ORGANIZATION_BLOCK "HardwareInterrupt"   // OB40, SCL, HardwareInterrupt
{ S7_Optimized_Access := 'TRUE' }
// stored: SetENOAutomatically false
   VAR_INPUT
      LADDR : HW_IO;   // Hardware identifier
      USI : Word;   // User structure identifier
      IChannel : USInt;   // Interrupt channel number
      EventType : Byte;   // EventType
      PointAddr : DWord;
   END_VAR
BEGIN
   REGION Description head
       //==================================================================================
       // POSALUX Swiss SA / (C) Copyright 2025
       //----------------------------------------------------------------------------------
       // Title: Hardware interrupt
       // Comment/Function: Executes when a relevant hardware event occurs
       // Author: Fabien WALDT
       // Engineering: TIA Portal v19
       //----------------------------------------------------------------------------------
       // Change log table:
       // Version  | Date     | Expert in charge | Changes applied
       //----------------------------------------------------------------------------------
       // 00.00.01 | 20250423 | WFA              | First released version
       //==================================================================================
   END_REGION

   REGION NCK Process IRT
       "LBP_NCKProcessIRT"(Flags => NULL);
   END_REGION
END_ORGANIZATION_BLOCK

ORGANIZATION_BLOCK "IO_AccessError"   // OB122, SCL, IOAccessError
{ S7_Optimized_Access := 'TRUE' }
// stored: SetENOAutomatically false
   VAR_INPUT
      BlockNr : UInt;   // Number of causing block
      Reaction : USInt;   // 0:ignore, 1:substitute, 2:skip
      Fault_ID : Byte;   // 16#42:reading, 16#43:writing
      BlockType : USInt;   // 16#01:OB, 16#02:FC, 16#03:FB, 16#04:SFC, 16#05:SFB, 16#06:DB: Type of block causing the error
      Area : USInt;   // 16#81:I, 16#82:Q: IO area where the IOaccess error occured
      DBNr : DB_ANY;   // Reserved for system
      Csg_OBNr : OB_ANY;   // Number of OB causing the error
      Csg_Prio : USInt;   // Priority of OB causing the error
      Width : USInt;   // 0:bit, 1:byte, 2:word, 3:dword, 4:lword
   END_VAR
BEGIN
   REGION Description head
       //==================================================================================
       // POSALUX Swiss SA / (C) Copyright 2025
       //----------------------------------------------------------------------------------
       // Title: IO_AccessError
       // Comment/Function: Executes whenever an error occurs while accessing data on a module
       // Author: Fabien WALDT
       // Engineering: TIA Portal v19
       //----------------------------------------------------------------------------------
       // Change log table:
       // Version  | Date     | Expert in charge | Changes applied
       //----------------------------------------------------------------------------------
       // 00.00.01 | 20250423 | WFA              | First released version
       //==================================================================================
   END_REGION
END_ORGANIZATION_BLOCK

ORGANIZATION_BLOCK "RackOrStationFailure"   // OB86, SCL, RackOrStationFailure
{ S7_Optimized_Access := 'TRUE' }
// stored: SetENOAutomatically false
   VAR_INPUT
      LADDR : HW_DEVICE;   // Hardware identifier
      Event_Class : Byte;   // Event class
      Fault_ID : Byte;   // Fault identifier
   END_VAR
BEGIN
   REGION Description head
       //==================================================================================
       // POSALUX Swiss SA / (C) Copyright 2025
       //----------------------------------------------------------------------------------
       // Title: Main
       // Comment/Function: Executes when the CPU detects the failure
       //                   or communication loss of a distributed rack or station
       // Author: Fabien WALDT
       // Engineering: TIA Portal v19
       //----------------------------------------------------------------------------------
       // Change log table:
       // Version  | Date     | Expert in charge | Changes applied
       //----------------------------------------------------------------------------------
       // 00.00.01 | 20250423 | WFA              | First released version
       //==================================================================================
   END_REGION
END_ORGANIZATION_BLOCK

ORGANIZATION_BLOCK "Startup"   // OB100, SCL, Startup
TITLE = "Complete Restart"
{ S7_Optimized_Access := 'TRUE' }
// stored: SetENOAutomatically false
   VAR_INPUT
      LostRetentive : Bool;   // True if retentive data are lost
      LostRTC : Bool;   // True if date and time are lost
   END_VAR
   VAR_TEMP
      tLastDateTime : DTL;
      tLasDateTimeSec : DInt;
      tActualDateTime : DTL;
      tActualDateTimeINT : DInt;
      tActualDateTimeSec : DInt;
   END_VAR
BEGIN
   REGION Description head
       //==================================================================================
       // POSALUX Swiss SA / (C) Copyright 2025
       //----------------------------------------------------------------------------------
       // Title: Startup
       // Comment/Function: Executes one time when the operating mode of the CPU changes from STOP to RUN
       // Author: Fabien WALDT
       // Engineering: TIA Portal v19
       //----------------------------------------------------------------------------------
       // Change log table:
       // Version  | Date     | Expert in charge | Changes applied
       //----------------------------------------------------------------------------------
       // 00.00.01 | 20250423 | WFA              | First released version
       //==================================================================================
   END_REGION

   REGION Safety Brake Test
       "LBP_AlarmMsgs".UserA[5].A70UUxx[12] := FALSE;  // Msg 700512 "SAFETY : THE BRAKE TEST IS NOT WORKING, PLEASE RESET"
   END_REGION

   REGION Config NC Panel
       "LBP_ConfigBP"(MCPNum := "LBP_ConfigData".MCPNum,
                      MCP1In := "MCP1_In",
                      MCP1Out := "MCP1_Out",
                      MCP1BusAdr := "LBP_ConfigData".MCP1BusAdr,
                      MCP1Timeout := "LBP_ConfigData".MCP1Timeout,
                      MCP2In := NULL,
                      MCP2Out := NULL,
                      MCP2BusAdr := "LBP_ConfigData".MCP2BusAdr,
                      MCP2Timeout := "LBP_ConfigData".MCP2Timeout,
                      MCP1Stop := "LBP_ConfigData".MCP1Stop,
                      MCP2Stop := "LBP_ConfigData".MCP2Stop,
                      MCP1NotSend := "LBP_ConfigData".MCP1NotSend,
                      MCP2NotSend := "LBP_ConfigData".MCP2NotSend,
                      MCPBusType := "LBP_ConfigData".MCPBusType,
                      HTIf := "LBP_ConfigData".HTIf,
                      HTIn := "LBP_ConfigData".HTIn,
                      HTOut := "LBP_ConfigData".HTOut,
                      HTAdr := "LBP_ConfigData".HTAdr,
                      HTStop := "LBP_ConfigData".HTStop,
                      HTNotSend := "LBP_ConfigData".HTNotSend,
                      NCCyclTimeout := "LBP_ConfigData".NCCyclTimeout,
                      NCRunupTimeout := "LBP_ConfigData".NCRunupTimeout,
                      ListMDecGrp := "LBP_ConfigData".ListMDecGrp,
                      MMCToIF := "LBP_ConfigData".MMCToIF,
                      HWheelMMC := "LBP_ConfigData".HWheelMMC,
                      MCP_IF_TCS := "LBP_ConfigData".MCP_IF_TCS,
                      ExtendChanAxMsg := "LBP_ConfigData".ExtendChanAxMsg,
                      HMIAxisSel := "LBP_ConfigData".HMIAxisSel,
                      DeactivateCtrlEnergy:=FALSE,
                      MsgUser := "LBP_ConfigData".MsgUser,
                      IRAuxfuT := "LBP_ConfigData".IRAuxfuT,
                      IRAuxfuH := "LBP_ConfigData".IRAuxfuH,
                      IRAuxfuE := "LBP_ConfigData".IRAuxfuE,
                      UserVersion := "LBP_ConfigData".UserVersionInfo,
                      OpKeyNum := "LBP_ConfigData".OpKeyNum,
                      Op1KeyIn := "LBP_ConfigData".Op1KeyIn,
                      Op1KeyOut := "LBP_ConfigData".Op1KeyOut,
                      Op1KeyBusAdr := "LBP_ConfigData".Op1KeyBusAdr,
                      Op2KeyIn := "LBP_ConfigData".Op2KeyIn,
                      Op2KeyOut := "LBP_ConfigData".Op2KeyOut,
                      Op2KeyBusAdr := "LBP_ConfigData".Op2KeyBusAdr,
                      Op1KeyStop := "LBP_ConfigData".Op1KeyStop,
                      Op2KeyStop := "LBP_ConfigData".Op2KeyStop,
                      Op1KeyNotSend := "LBP_ConfigData".Op1KeyNotSend,
                      Op2KeyNotSend := "LBP_ConfigData".Op2KeyNotSend,
                      OpUnitCommId := "LBP_ConfigData".OpUnitCommId,
                      OpUnitInterfaceId := "LBP_ConfigData".OpUnitInterfaceId,
                      MCP1ConnectionId := "LBP_ConfigData".MCP1ConnectionId,
                      MCP2ConnectionId := "LBP_ConfigData".MCP2ConnectionId,
                      HTConnectionId := "LBP_ConfigData".HTConnectionId,
                      Op1KeyConnectionId := "LBP_ConfigData".Op1KeyConnectionId,
                      Op2KeyConnectionId := "LBP_ConfigData".Op2KeyConnectionId,
                      IdentConnectionId := "LBP_ConfigData".IdentConnectionId,
                      MCP1LocalUdpPort := "LBP_ConfigData".MCP1LocalUdpPort,
                      MCP2LocalUdpPort := "LBP_ConfigData".MCP2LocalUdpPort,
                      HTLocalUdpPort := "LBP_ConfigData".HTLocalUdpPort,
                      Op1KeyLocalUdpPort := "LBP_ConfigData".Op1KeyLocalUdpPort,
                      Op2KeyLocalUdpPort := "LBP_ConfigData".Op2KeyLocalUdpPort,
                      IdentLocalUdpPort := "LBP_ConfigData".IdentLocalUdpPort,
                      MaxModeGroup => "LBP_ConfigData".MaxModeGroup,
                      MaxChan => "LBP_ConfigData".MaxChan,
                      MaxAxis => "LBP_ConfigData".MaxAxis,
                      ActiveChan => "LBP_ConfigData".ActiveChan,
                      ActiveAxis => "LBP_ConfigData".ActiveAxis,
                      MaxNumUserDataInt => "LBP_ConfigData".MaxNumUserDataInt,
                      MaxNumUserDataHex => "LBP_ConfigData".MaxNumUserDataHex,
                      MaxNumUserDataReal => "LBP_ConfigData".MaxNumUserDataReal,
                      UserDataIntArray => NULL,
                      UserDataHexArray => NULL,
                      UserDataRealArray => NULL,
                      TMMagazines => NULL);
   END_REGION

   REGION RAZ Shutdown variables
       "LBP_AlarmMsgs".UserA[04].A70UUxx[05] := FALSE;  // Msg 700405 "UPS power failure"
       "LBP_AlarmMsgs".UserA[04].A70UUxx[41] := FALSE;  // Msg 700441 "Machine stop process completed. Turn off the machine using the main switch"
       "LBP_AlarmMsgs".UserA[04].A70UUxx[42] := FALSE;  // Msg 700442 "The machine stop process has started..."
       "LBP_AlarmMsgs".UserA[04].A70UUxx[20] := FALSE;  // Msg 700420 "Timeout shutdown. Please turn off manually"
       "LBP_AlarmMsgs".UserA[04].A70UUxx[21] := FALSE;  // Msg 700421 "The laser is still on. Please turn it off manually"
       "LBP_AlarmMsgs".UserA[04].A70UUxx[22] := FALSE;  // Msg 700422 "Laser status unknown. Turn it off on left PC then wait for the machine's shutdown"
       "LBP_AlarmMsgs".UserA[04].A70UUxx[23] := FALSE;  // Msg 700423 "Power failure. The machine stop process has started…"

       "DB_Machineshutdown_UPS".sShutDownPCRequest    := 0;
       "DB_Machineshutdown_UPS".sShutDownPCResponse   := 0;
   END_REGION
END_ORGANIZATION_BLOCK

FUNCTION_BLOCK "FB_Nouveau"   // FB91, SCL
{ S7_Optimized_Access := 'TRUE' }
// stored: MemoryReserve 100, SetENOAutomatically false
   VAR
      "#sExtLoadUnloadTimer1" : TON_TIME;
      "#sExtLoadUnloadTimer2" { S7_SetPoint := 'True'} : TON_TIME;
   END_VAR
BEGIN
   REGION Ext Load/Unload Time
       // Necessaire pour Dry Run
       // #sExtLoadUnloadTimer1(IN := "DB_LoaderShuttle1".sExtLoadUnload.sCurrent_Step_NB = 50
       //                       OR "DB_LoaderShuttle1".sExtLoadUnload.sCurrent_Step_NB = 80
       //                       OR "DB_LoaderShuttle1".sExtLoadUnload.sCurrent_Step_NB = 110,
       //                       PT := t#3s);
       // "DB_SonplasMain".sSonplasLoader.iPartInShuttle1Finished := #sExtLoadUnloadTimer1.Q;

       // #sExtLoadUnloadTimer2(IN := "DB_LoaderShuttle2".sExtLoadUnload.sCurrent_Step_NB = 50
       //                       OR "DB_LoaderShuttle2".sExtLoadUnload.sCurrent_Step_NB = 80
       //                       OR "DB_LoaderShuttle2".sExtLoadUnload.sCurrent_Step_NB = 110,
       //                       PT := t#3s);
       // "DB_SonplasMain".sSonplasLoader.iPartInShuttle2Finished := #sExtLoadUnloadTimer2.Q;
   END_REGION
END_FUNCTION_BLOCK

FUNCTION_BLOCK "FB_Counter"   // FB40, SCL
{ S7_Optimized_Access := 'TRUE' }
// stored: MemoryReserve 100, SetENOAutomatically false
   VAR_INPUT
      iIncrement : Bool;
      iReset : Bool;
      iLimit : UDInt;
   END_VAR
   VAR_OUTPUT
      oLimitReached : Bool;
   END_VAR
   VAR
      sRT_Increment { ExternalAccessible := 'False'; ExternalVisible := 'False'; ExternalWritable := 'False'} : R_TRIG;
      sCounter { S7_SetPoint := 'True'} : UDInt;
      sCounterNoReset : UDInt;
   END_VAR
BEGIN
   REGION Description header 
       //==================================================================================
       // POSALUX Swiss SA / (C) Copyright 2025
       //----------------------------------------------------------------------------------
       // Title: FB_Counter
       // Comment/Function: This function allows:
       //                      - Counting Pulse
       //
       // Author: Fabien Waldt
       // Engineering: TIA Portal v19
       //----------------------------------------------------------------------------------
       // Change log table:
       // Version  | Date     | Expert in charge | Changes applied
       // ---------|----------|------------------|------------------------------------
       // 00.00.01 | 20250718 | WFA              | First released version
       // ==================================================================================
   END_REGION

   REGION Counter Reset
       IF #iReset THEN
           #sCounter := 0;
       END_IF;

       IF #sCounterNoReset >= 4294967295 THEN
           #sCounterNoReset := 0;
       END_IF;
   END_REGION

   REGION Counter Increment
       #sRT_Increment(CLK := #iIncrement);

       IF #sRT_Increment.Q THEN
           #sCounter := #sCounter + 1;
           #sCounterNoReset := #sCounterNoReset + 1;
       END_IF;
   END_REGION ;

   REGION Limit Reached
       #oLimitReached := #sCounter >= #iLimit;
   END_REGION ;
END_FUNCTION_BLOCK

FUNCTION "FC_CheckTimeout" : Void   // FC34, SCL
{ S7_Optimized_Access := 'TRUE' }
// stored: SetENOAutomatically false
   VAR_INPUT
      iCondition : Bool;
      iTime : Time;
   END_VAR
   VAR_OUTPUT
      oTimeoutOccurred : Bool;
   END_VAR
   VAR_IN_OUT
      ioTimer : TON_TIME;
   END_VAR
BEGIN
   REGION Description header 
       //==================================================================================
       // POSALUX Swiss SA / (C) Copyright 2025
       //----------------------------------------------------------------------------------
       // Title: CheckTimeout
       // Comment/Function: Start a Timeout control according conditions
       //                   Set a bit at the end of the timer
       // Author: Fabien WALDT
       // Engineering: TIA Portal v17
       //----------------------------------------------------------------------------------
       // Change log table:
       // Version  | Date     | Expert in charge | Changes applied
       // ---------|----------|------------------|-----------------------------------------
       // 00.00.01 | 20250423 | WFA              | First released version
       // =================================================================================
   END_REGION
   // Configuration du timer
   #ioTimer.PT := #iTime;

   // Activation du timer si la condition est vraie
   #ioTimer.IN := #iCondition;

   // Vérification du timeout
   IF #ioTimer.Q THEN
       #oTimeoutOccurred := true;
   ELSIF "MCP1_In".reset THEN
       #oTimeoutOccurred := false;
   END_IF;
END_FUNCTION

FUNCTION_BLOCK "Main_Safety_RTG1"   // FB30, F_LAD
{ S7_Optimized_Access := 'TRUE' }
// ============================================================================
// // POSALUX Swiss SA / (C) Copyright 2024
// //----------------------------------------------------------------------------------
// // Title: Programme Principale Safety
// // Comment/Function: 
// //
// // Author: Olivier Heim
// // Engineering: TIA Portal v17
// //----------------------------------------------------------------------------------
// // Change log table:
// // Version   | Date            | Expert in charge | Changes applied
// // -----------------|---------------------|--------------------------------|------------------------------------
// // 00.00.01 | 20241218 | HOL                        | First released version
// // -----------------|---------------------|--------------------------------|------------------------------------
// // 01.01.00 | 20241218 | FMI                         | General improves
// / ============================================================================
// stored: AutoNumber false
   VAR
      sSupplyPower : Bool;
      sAckEmergencyStop : Bool;
      sAckFdbPowMach : Bool;
      sAckFdbBW_LoaderEstopRelay : Bool;
      sAckFdbSonplasDoorClosedRelay : Bool;
      ESTOP1_Instance : ESTOP1;
      FDBACK_PowerMachine : FDBACK;
      FDBACK_BW_LoaderEstopRelay : FDBACK;
      FDBACK_SonplasDoorClosedRelay : FDBACK;
      DB_ACK_GL : ACK_GL;
   END_VAR
BEGIN

REGION Network 1: Transfer DataToSafety to DataToSafety F
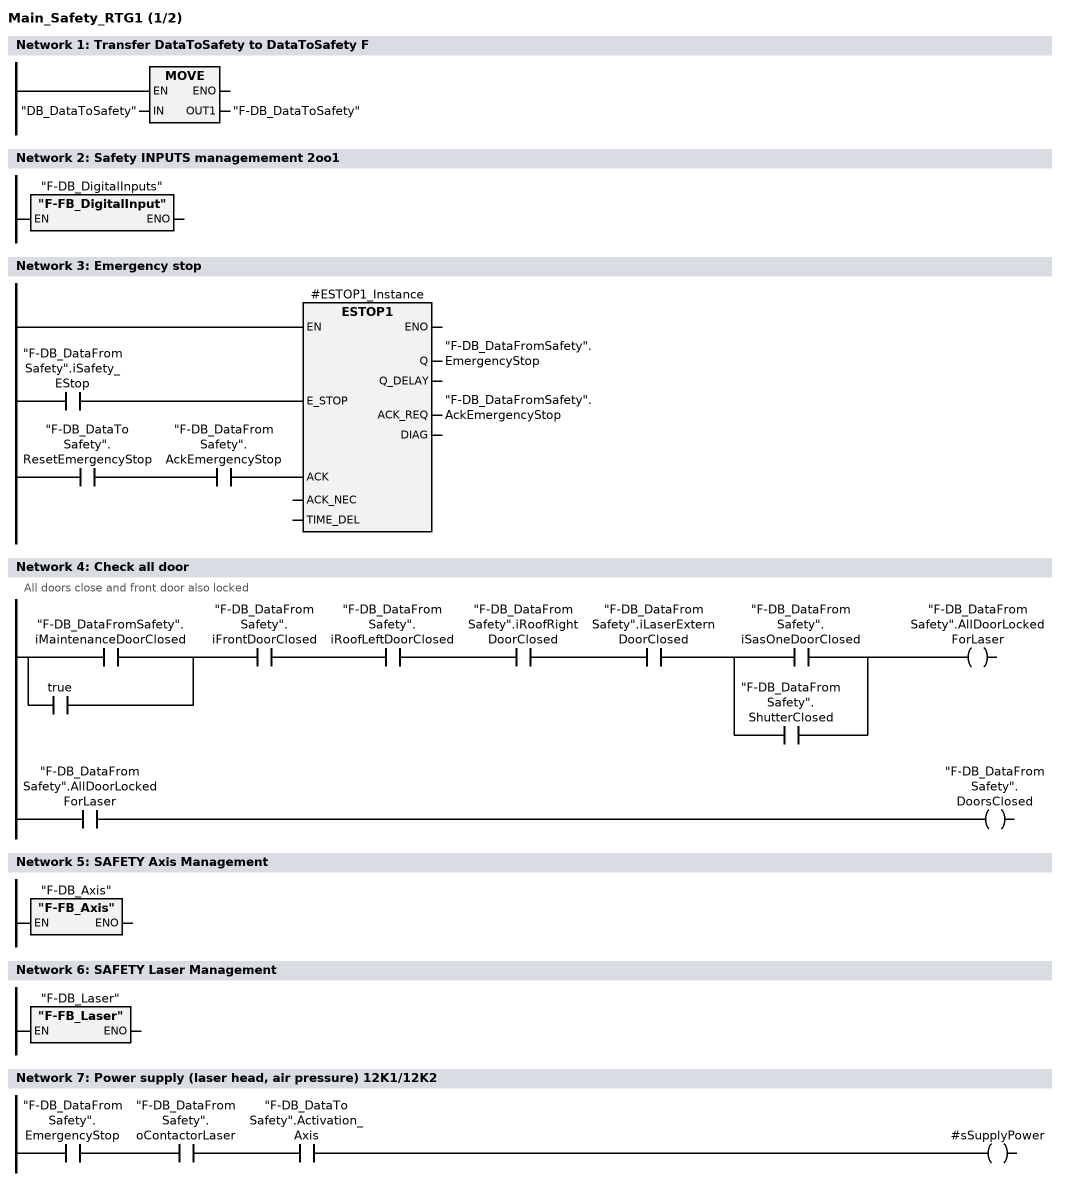
   RUNG wire#powerrail
      { S7_GenerateENO := "TRUE" } Move(in := "DB_DataToSafety", out1 => "F-DB_DataToSafety")
   END_RUNG
   // the same network as SCL:
   "F-DB_DataToSafety" := "DB_DataToSafety";
END_REGION

REGION Network 2: Safety INPUTS managemement 2oo1
   RUNG wire#powerrail
      "F-DB_DigitalInputs"()
   END_RUNG
   // the same network as SCL:
   "F-DB_DigitalInputs"();   // "F-FB_DigitalInput"
END_REGION

REGION Network 3: Emergency stop
   RUNG wire#powerrail
      #ESTOP1_Instance.ESTOP1(E_STOP := wire#w1, ACK := wire#w2, ACK_NEC :=, TIME_DEL :=, Q => "F-DB_DataFromSafety".EmergencyStop, Q_DELAY =>, ACK_REQ => "F-DB_DataFromSafety".AckEmergencyStop, DIAG =>)
   END_RUNG
   RUNG wire#powerrail
      Contact( "F-DB_DataFromSafety".iSafety_EStop )
   END_RUNG wire#w1
   RUNG wire#powerrail
      Contact( "F-DB_DataToSafety".ResetEmergencyStop )
      Contact( "F-DB_DataFromSafety".AckEmergencyStop )
   END_RUNG wire#w2
   // the same network as SCL:
   #ESTOP1_Instance(E_STOP := "F-DB_DataFromSafety".iSafety_EStop,   // ESTOP1
                    ACK := "F-DB_DataToSafety".ResetEmergencyStop AND "F-DB_DataFromSafety".AckEmergencyStop,
                    Q => "F-DB_DataFromSafety".EmergencyStop,
                    ACK_REQ => "F-DB_DataFromSafety".AckEmergencyStop);
END_REGION

REGION Network 4: Check all door
   // All doors close and front door also locked
   RUNG wire#powerrail
      Contact( "F-DB_DataFromSafety".iMaintenanceDoorClosed )
      wire#w1
      Contact( "F-DB_DataFromSafety".iFrontDoorClosed )
      Contact( "F-DB_DataFromSafety".iRoofLeftDoorClosed )
      Contact( "F-DB_DataFromSafety".iRoofRightDoorClosed )
      Contact( "F-DB_DataFromSafety".iLaserExternDoorClosed )
      wire#w2
      Contact( "F-DB_DataFromSafety".iSasOneDoorClosed )
      wire#w3
      Coil( "F-DB_DataFromSafety".AllDoorLockedForLaser )
   END_RUNG
   RUNG wire#powerrail
      Contact( true )
   END_RUNG wire#w1
   RUNG wire#w2
      Contact( "F-DB_DataFromSafety".ShutterClosed )
   END_RUNG wire#w3
   RUNG wire#powerrail
      Contact( "F-DB_DataFromSafety".AllDoorLockedForLaser )
      Coil( "F-DB_DataFromSafety".DoorsClosed )
   END_RUNG
   // the same network as SCL:
   "F-DB_DataFromSafety".AllDoorLockedForLaser := ("F-DB_DataFromSafety".iMaintenanceDoorClosed OR true) AND "F-DB_DataFromSafety".iFrontDoorClosed AND "F-DB_DataFromSafety".iRoofLeftDoorClosed AND "F-DB_DataFromSafety".iRoofRightDoorClosed AND "F-DB_DataFromSafety".iLaserExternDoorClosed AND ("F-DB_DataFromSafety".iSasOneDoorClosed OR "F-DB_DataFromSafety".ShutterClosed);
   "F-DB_DataFromSafety".DoorsClosed := "F-DB_DataFromSafety".AllDoorLockedForLaser;
END_REGION

REGION Network 5: SAFETY Axis Management
   RUNG wire#powerrail
      "F-DB_Axis"()
   END_RUNG
   // the same network as SCL:
   "F-DB_Axis"();   // "F-FB_Axis"
END_REGION

REGION Network 6: SAFETY Laser Management
   RUNG wire#powerrail
      "F-DB_Laser"()
   END_RUNG
   // the same network as SCL:
   "F-DB_Laser"();   // "F-FB_Laser"
END_REGION

REGION Network 7: Power supply (laser head, air pressure) 12K1/12K2
   RUNG wire#powerrail
      Contact( "F-DB_DataFromSafety".EmergencyStop )
      Contact( "F-DB_DataFromSafety".oContactorLaser )
      Contact( "F-DB_DataToSafety".Activation_Axis )
      Coil( #sSupplyPower )
   END_RUNG
   // the same network as SCL:
   #sSupplyPower := "F-DB_DataFromSafety".EmergencyStop AND "F-DB_DataFromSafety".oContactorLaser AND "F-DB_DataToSafety".Activation_Axis;
END_REGION

REGION Network 8: Check feed back power supply
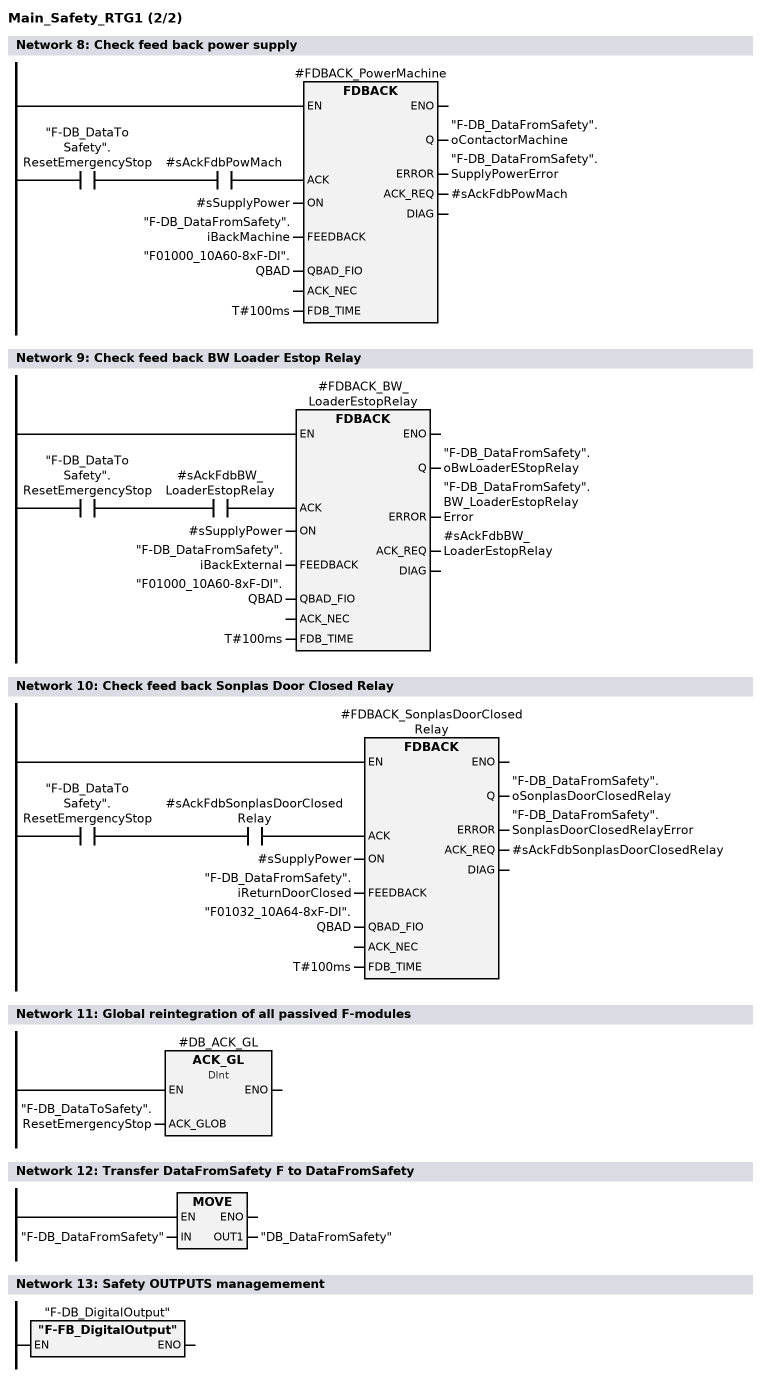
   RUNG wire#powerrail
      #FDBACK_PowerMachine.FDBACK(ACK := wire#w1, ON := #sSupplyPower, FEEDBACK := "F-DB_DataFromSafety".iBackMachine, QBAD_FIO := "F01000_10A60-8xF-DI".QBAD, ACK_NEC :=, FDB_TIME := T#100ms, Q => "F-DB_DataFromSafety".oContactorMachine, ERROR => "F-DB_DataFromSafety".SupplyPowerError, ACK_REQ => #sAckFdbPowMach, DIAG =>)
   END_RUNG
   RUNG wire#powerrail
      Contact( "F-DB_DataToSafety".ResetEmergencyStop )
      Contact( #sAckFdbPowMach )
   END_RUNG wire#w1
   // the same network as SCL:
   #FDBACK_PowerMachine(ACK := "F-DB_DataToSafety".ResetEmergencyStop AND #sAckFdbPowMach,   // FDBACK
                        ON := #sSupplyPower,
                        FEEDBACK := "F-DB_DataFromSafety".iBackMachine,
                        QBAD_FIO := "F01000_10A60-8xF-DI".QBAD,
                        FDB_TIME := T#100ms,
                        Q => "F-DB_DataFromSafety".oContactorMachine,
                        ERROR => "F-DB_DataFromSafety".SupplyPowerError,
                        ACK_REQ => #sAckFdbPowMach);
END_REGION

REGION Network 9: Check feed back BW Loader Estop Relay
   RUNG wire#powerrail
      #FDBACK_BW_LoaderEstopRelay.FDBACK(ACK := wire#w1, ON := #sSupplyPower, FEEDBACK := "F-DB_DataFromSafety".iBackExternal, QBAD_FIO := "F01000_10A60-8xF-DI".QBAD, ACK_NEC :=, FDB_TIME := T#100ms, Q => "F-DB_DataFromSafety".oBwLoaderEStopRelay, ERROR => "F-DB_DataFromSafety".BW_LoaderEstopRelayError, ACK_REQ => #sAckFdbBW_LoaderEstopRelay, DIAG =>)
   END_RUNG
   RUNG wire#powerrail
      Contact( "F-DB_DataToSafety".ResetEmergencyStop )
      Contact( #sAckFdbBW_LoaderEstopRelay )
   END_RUNG wire#w1
   // the same network as SCL:
   #FDBACK_BW_LoaderEstopRelay(ACK := "F-DB_DataToSafety".ResetEmergencyStop AND #sAckFdbBW_LoaderEstopRelay,   // FDBACK
                           ON := #sSupplyPower,
                           FEEDBACK := "F-DB_DataFromSafety".iBackExternal,
                           QBAD_FIO := "F01000_10A60-8xF-DI".QBAD,
                           FDB_TIME := T#100ms,
                           Q => "F-DB_DataFromSafety".oBwLoaderEStopRelay,
                           ERROR => "F-DB_DataFromSafety".BW_LoaderEstopRelayError,
                           ACK_REQ => #sAckFdbBW_LoaderEstopRelay);
END_REGION

REGION Network 10: Check feed back Sonplas Door Closed Relay
   RUNG wire#powerrail
      #FDBACK_SonplasDoorClosedRelay.FDBACK(ACK := wire#w1, ON := #sSupplyPower, FEEDBACK := "F-DB_DataFromSafety".iReturnDoorClosed, QBAD_FIO := "F01032_10A64-8xF-DI".QBAD, ACK_NEC :=, FDB_TIME := T#100ms, Q => "F-DB_DataFromSafety".oSonplasDoorClosedRelay, ERROR => "F-DB_DataFromSafety".SonplasDoorClosedRelayError, ACK_REQ => #sAckFdbSonplasDoorClosedRelay, DIAG =>)
   END_RUNG
   RUNG wire#powerrail
      Contact( "F-DB_DataToSafety".ResetEmergencyStop )
      Contact( #sAckFdbSonplasDoorClosedRelay )
   END_RUNG wire#w1
   // the same network as SCL:
   #FDBACK_SonplasDoorClosedRelay(ACK := "F-DB_DataToSafety".ResetEmergencyStop AND #sAckFdbSonplasDoorClosedRelay,   // FDBACK
                           ON := #sSupplyPower,
                           FEEDBACK := "F-DB_DataFromSafety".iReturnDoorClosed,
                           QBAD_FIO := "F01032_10A64-8xF-DI".QBAD,
                           FDB_TIME := T#100ms,
                           Q => "F-DB_DataFromSafety".oSonplasDoorClosedRelay,
                           ERROR => "F-DB_DataFromSafety".SonplasDoorClosedRelayError,
                           ACK_REQ => #sAckFdbSonplasDoorClosedRelay);
END_REGION

REGION Network 11: Global reintegration of all passived F-modules
   RUNG wire#powerrail
      { S7_Templates := "codedbool_type := DInt" } #DB_ACK_GL.ACK_GL(ACK_GLOB := "F-DB_DataToSafety".ResetEmergencyStop)
   END_RUNG
   // the same network as SCL:
   #DB_ACK_GL(ACK_GLOB := "F-DB_DataToSafety".ResetEmergencyStop);   // ACK_GL
END_REGION

REGION Network 12: Transfer DataFromSafety F to DataFromSafety
   RUNG wire#powerrail
      { S7_GenerateENO := "TRUE" } Move(in := "F-DB_DataFromSafety", out1 => "DB_DataFromSafety")
   END_RUNG
   // the same network as SCL:
   "DB_DataFromSafety" := "F-DB_DataFromSafety";
END_REGION

REGION Network 13: Safety OUTPUTS managemement
   RUNG wire#powerrail
      "F-DB_DigitalOutput"()
   END_RUNG
   // the same network as SCL:
   "F-DB_DigitalOutput"();   // "F-FB_DigitalOutput"
END_REGION
END_FUNCTION_BLOCK

FUNCTION_BLOCK "F-FB_DigitalInput"   // FB110, F_LAD
{ S7_Optimized_Access := 'TRUE' }
// stored: AutoNumber false
   VAR
      sSafety_EStop : EV1oo2DI;
      sKeySettingMode : EV1oo2DI;
      sKeySettingLaser : EV1oo2DI;
      sMaintenanceDoorClosed : EV1oo2DI;
      sFrontDoorClosed : EV1oo2DI;
      sEmergencyStopPowerLaser : EV1oo2DI;
      sRoofLeftDoorClosed : EV1oo2DI;
      sKeyLaserON : EV1oo2DI;
      sLaserExternDoorClosed : EV1oo2DI;
      sSasOneDoorClosed : EV1oo2DI;
      sBwLoaderDoorClosed : EV1oo2DI;
      sRoofRightDoorClosed : EV1oo2DI;
      sSonplas_EStop : EV1oo2DI;
      sBwLoader_EStop : EV1oo2DI;
      sSonplasDoorClosed : EV1oo2DI;
      sAck_iSafety_EStop { ExternalAccessible := 'False'; ExternalVisible := 'False'; ExternalWritable := 'False'} : Bool;
      sAck_iKeySettingMode { ExternalAccessible := 'False'; ExternalVisible := 'False'; ExternalWritable := 'False'} : Bool;
      sAck_iKeySettingLaser { ExternalAccessible := 'False'; ExternalVisible := 'False'; ExternalWritable := 'False'} : Bool;
      sAck_iMaintenanceDoorClosed { ExternalAccessible := 'False'; ExternalVisible := 'False'; ExternalWritable := 'False'} : Bool;
      sAck_iFrontDoorClosed { ExternalAccessible := 'False'; ExternalVisible := 'False'; ExternalWritable := 'False'} : Bool;
      sAck_iEmergencyStopPowerLaser { ExternalAccessible := 'False'; ExternalVisible := 'False'; ExternalWritable := 'False'} : Bool;
      sAck_iRoofLeftDoorClosed { ExternalAccessible := 'False'; ExternalVisible := 'False'; ExternalWritable := 'False'} : Bool;
      sAck_iKeyLaserON { ExternalAccessible := 'False'; ExternalVisible := 'False'; ExternalWritable := 'False'} : Bool;
      sAck_iLaserExternDoorClosed : Bool;
      sAck_iSasOneDoorClosed { ExternalAccessible := 'False'; ExternalVisible := 'False'; ExternalWritable := 'False'} : Bool;
      sAck_iBwLoaderDoorClosed : Bool;
      sAck_iRoofRightDoorClosed { ExternalAccessible := 'False'; ExternalVisible := 'False'; ExternalWritable := 'False'} : Bool;
      sAck_iSonplas_EStop : Bool;
      sAck_iBwLoader_EStop : Bool;
      sAck_iSonplasDoorClosed { ExternalAccessible := 'False'; ExternalVisible := 'False'; ExternalWritable := 'False'} : Bool;
   END_VAR
BEGIN

REGION Network 1: Safety EStop
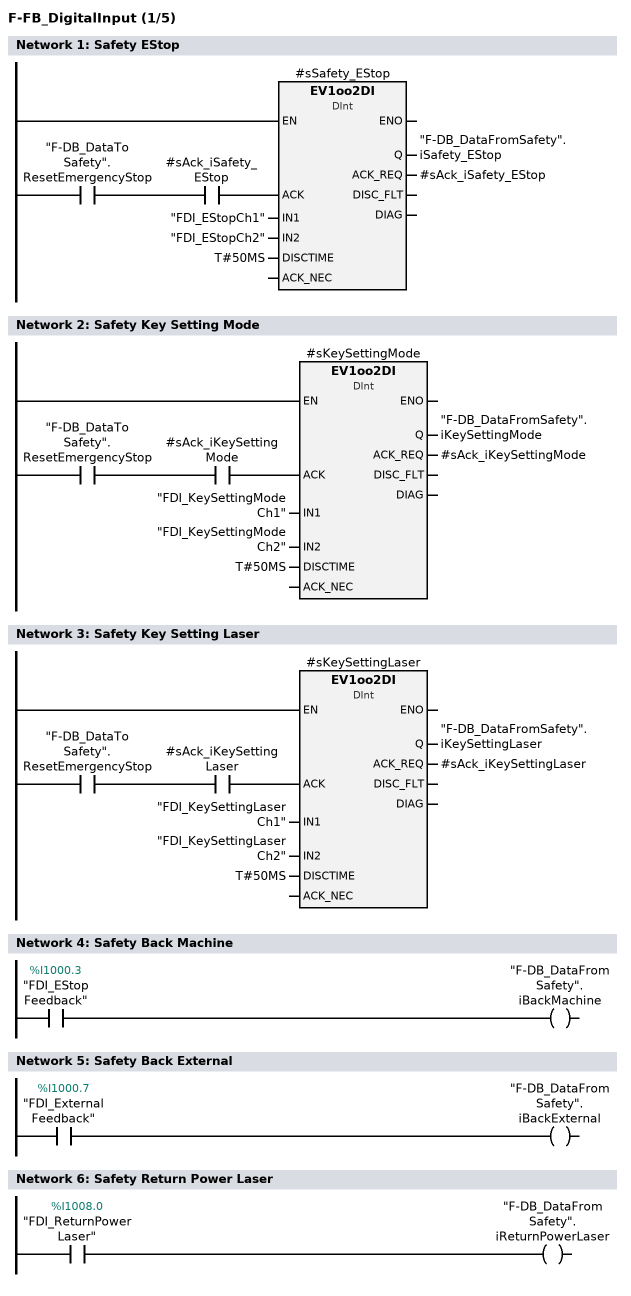
   RUNG wire#powerrail
      { S7_Templates := "codedbool_type := DInt" } #sSafety_EStop.EV1oo2DI(ACK := wire#w1, IN1 := "FDI_EStopCh1", IN2 := "FDI_EStopCh2", DISCTIME := T#50MS, ACK_NEC :=, Q => "F-DB_DataFromSafety".iSafety_EStop, ACK_REQ => #sAck_iSafety_EStop, DISC_FLT =>, DIAG =>)
   END_RUNG
   RUNG wire#powerrail
      Contact( "F-DB_DataToSafety".ResetEmergencyStop )
      Contact( #sAck_iSafety_EStop )
   END_RUNG wire#w1
   // the same network as SCL:
   #sSafety_EStop(ACK := "F-DB_DataToSafety".ResetEmergencyStop AND #sAck_iSafety_EStop,   // EV1oo2DI
                  IN1 := "FDI_EStopCh1",
                  IN2 := "FDI_EStopCh2",
                  DISCTIME := T#50MS,
                  Q => "F-DB_DataFromSafety".iSafety_EStop,
                  ACK_REQ => #sAck_iSafety_EStop);
END_REGION

REGION Network 2: Safety Key Setting Mode
   RUNG wire#powerrail
      { S7_Templates := "codedbool_type := DInt" } #sKeySettingMode.EV1oo2DI(ACK := wire#w1, IN1 := "FDI_KeySettingModeCh1", IN2 := "FDI_KeySettingModeCh2", DISCTIME := T#50MS, ACK_NEC :=, Q => "F-DB_DataFromSafety".iKeySettingMode, ACK_REQ => #sAck_iKeySettingMode, DISC_FLT =>, DIAG =>)
   END_RUNG
   RUNG wire#powerrail
      Contact( "F-DB_DataToSafety".ResetEmergencyStop )
      Contact( #sAck_iKeySettingMode )
   END_RUNG wire#w1
   // the same network as SCL:
   #sKeySettingMode(ACK := "F-DB_DataToSafety".ResetEmergencyStop AND #sAck_iKeySettingMode,   // EV1oo2DI
                    IN1 := "FDI_KeySettingModeCh1",
                    IN2 := "FDI_KeySettingModeCh2",
                    DISCTIME := T#50MS,
                    Q => "F-DB_DataFromSafety".iKeySettingMode,
                    ACK_REQ => #sAck_iKeySettingMode);
END_REGION

REGION Network 3: Safety Key Setting Laser
   RUNG wire#powerrail
      { S7_Templates := "codedbool_type := DInt" } #sKeySettingLaser.EV1oo2DI(ACK := wire#w1, IN1 := "FDI_KeySettingLaserCh1", IN2 := "FDI_KeySettingLaserCh2", DISCTIME := T#50MS, ACK_NEC :=, Q => "F-DB_DataFromSafety".iKeySettingLaser, ACK_REQ => #sAck_iKeySettingLaser, DISC_FLT =>, DIAG =>)
   END_RUNG
   RUNG wire#powerrail
      Contact( "F-DB_DataToSafety".ResetEmergencyStop )
      Contact( #sAck_iKeySettingLaser )
   END_RUNG wire#w1
   // the same network as SCL:
   #sKeySettingLaser(ACK := "F-DB_DataToSafety".ResetEmergencyStop AND #sAck_iKeySettingLaser,   // EV1oo2DI
                     IN1 := "FDI_KeySettingLaserCh1",
                     IN2 := "FDI_KeySettingLaserCh2",
                     DISCTIME := T#50MS,
                     Q => "F-DB_DataFromSafety".iKeySettingLaser,
                     ACK_REQ => #sAck_iKeySettingLaser);
END_REGION

REGION Network 4: Safety Back Machine
   RUNG wire#powerrail
      Contact( "FDI_EStopFeedback" )
      Coil( "F-DB_DataFromSafety".iBackMachine )
   END_RUNG
   // the same network as SCL:
   "F-DB_DataFromSafety".iBackMachine := "FDI_EStopFeedback";
END_REGION

REGION Network 5: Safety Back External
   RUNG wire#powerrail
      Contact( "FDI_ExternalFeedback" )
      Coil( "F-DB_DataFromSafety".iBackExternal )
   END_RUNG
   // the same network as SCL:
   "F-DB_DataFromSafety".iBackExternal := "FDI_ExternalFeedback";
END_REGION

REGION Network 6: Safety Return Power Laser
   RUNG wire#powerrail
      Contact( "FDI_ReturnPowerLaser" )
      Coil( "F-DB_DataFromSafety".iReturnPowerLaser )
   END_RUNG
   // the same network as SCL:
   "F-DB_DataFromSafety".iReturnPowerLaser := "FDI_ReturnPowerLaser";
END_REGION

REGION Network 7: Safety Maintenance Door Closed
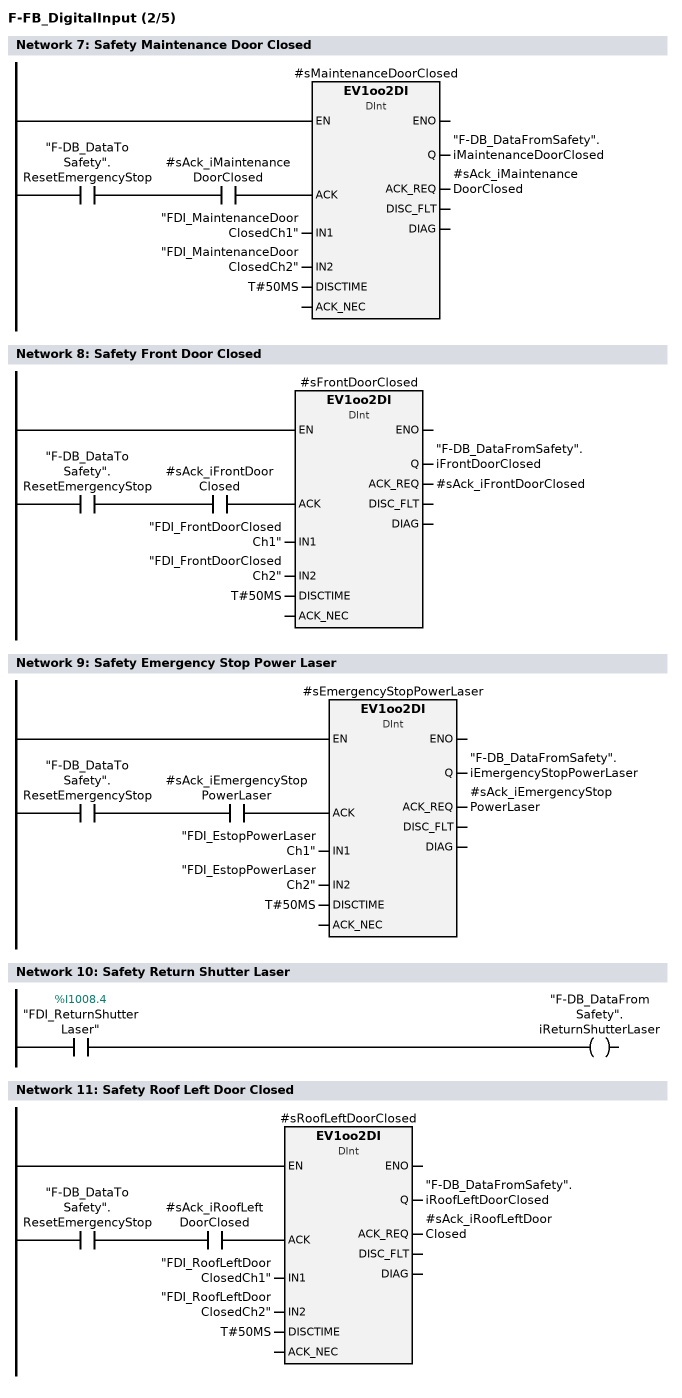
   RUNG wire#powerrail
      { S7_Templates := "codedbool_type := DInt" } #sMaintenanceDoorClosed.EV1oo2DI(ACK := wire#w1, IN1 := "FDI_MaintenanceDoorClosedCh1", IN2 := "FDI_MaintenanceDoorClosedCh2", DISCTIME := T#50MS, ACK_NEC :=, Q => "F-DB_DataFromSafety".iMaintenanceDoorClosed, ACK_REQ => #sAck_iMaintenanceDoorClosed, DISC_FLT =>, DIAG =>)
   END_RUNG
   RUNG wire#powerrail
      Contact( "F-DB_DataToSafety".ResetEmergencyStop )
      Contact( #sAck_iMaintenanceDoorClosed )
   END_RUNG wire#w1
   // the same network as SCL:
   #sMaintenanceDoorClosed(ACK := "F-DB_DataToSafety".ResetEmergencyStop AND #sAck_iMaintenanceDoorClosed,   // EV1oo2DI
                           IN1 := "FDI_MaintenanceDoorClosedCh1",
                           IN2 := "FDI_MaintenanceDoorClosedCh2",
                           DISCTIME := T#50MS,
                           Q => "F-DB_DataFromSafety".iMaintenanceDoorClosed,
                           ACK_REQ => #sAck_iMaintenanceDoorClosed);
END_REGION

REGION Network 8: Safety Front Door Closed
   RUNG wire#powerrail
      { S7_Templates := "codedbool_type := DInt" } #sFrontDoorClosed.EV1oo2DI(ACK := wire#w1, IN1 := "FDI_FrontDoorClosedCh1", IN2 := "FDI_FrontDoorClosedCh2", DISCTIME := T#50MS, ACK_NEC :=, Q => "F-DB_DataFromSafety".iFrontDoorClosed, ACK_REQ => #sAck_iFrontDoorClosed, DISC_FLT =>, DIAG =>)
   END_RUNG
   RUNG wire#powerrail
      Contact( "F-DB_DataToSafety".ResetEmergencyStop )
      Contact( #sAck_iFrontDoorClosed )
   END_RUNG wire#w1
   // the same network as SCL:
   #sFrontDoorClosed(ACK := "F-DB_DataToSafety".ResetEmergencyStop AND #sAck_iFrontDoorClosed,   // EV1oo2DI
                     IN1 := "FDI_FrontDoorClosedCh1",
                     IN2 := "FDI_FrontDoorClosedCh2",
                     DISCTIME := T#50MS,
                     Q => "F-DB_DataFromSafety".iFrontDoorClosed,
                     ACK_REQ => #sAck_iFrontDoorClosed);
END_REGION

REGION Network 9: Safety Emergency Stop Power Laser
   RUNG wire#powerrail
      { S7_Templates := "codedbool_type := DInt" } #sEmergencyStopPowerLaser.EV1oo2DI(ACK := wire#w1, IN1 := "FDI_EstopPowerLaserCh1", IN2 := "FDI_EstopPowerLaserCh2", DISCTIME := T#50MS, ACK_NEC :=, Q => "F-DB_DataFromSafety".iEmergencyStopPowerLaser, ACK_REQ => #sAck_iEmergencyStopPowerLaser, DISC_FLT =>, DIAG =>)
   END_RUNG
   RUNG wire#powerrail
      Contact( "F-DB_DataToSafety".ResetEmergencyStop )
      Contact( #sAck_iEmergencyStopPowerLaser )
   END_RUNG wire#w1
   // the same network as SCL:
   #sEmergencyStopPowerLaser(ACK := "F-DB_DataToSafety".ResetEmergencyStop AND #sAck_iEmergencyStopPowerLaser,   // EV1oo2DI
                           IN1 := "FDI_EstopPowerLaserCh1",
                           IN2 := "FDI_EstopPowerLaserCh2",
                           DISCTIME := T#50MS,
                           Q => "F-DB_DataFromSafety".iEmergencyStopPowerLaser,
                           ACK_REQ => #sAck_iEmergencyStopPowerLaser);
END_REGION

REGION Network 10: Safety Return Shutter Laser
   RUNG wire#powerrail
      Contact( "FDI_ReturnShutterLaser" )
      Coil( "F-DB_DataFromSafety".iReturnShutterLaser )
   END_RUNG
   // the same network as SCL:
   "F-DB_DataFromSafety".iReturnShutterLaser := "FDI_ReturnShutterLaser";
END_REGION

REGION Network 11: Safety Roof Left Door Closed
   RUNG wire#powerrail
      { S7_Templates := "codedbool_type := DInt" } #sRoofLeftDoorClosed.EV1oo2DI(ACK := wire#w1, IN1 := "FDI_RoofLeftDoorClosedCh1", IN2 := "FDI_RoofLeftDoorClosedCh2", DISCTIME := T#50MS, ACK_NEC :=, Q => "F-DB_DataFromSafety".iRoofLeftDoorClosed, ACK_REQ => #sAck_iRoofLeftDoorClosed, DISC_FLT =>, DIAG =>)
   END_RUNG
   RUNG wire#powerrail
      Contact( "F-DB_DataToSafety".ResetEmergencyStop )
      Contact( #sAck_iRoofLeftDoorClosed )
   END_RUNG wire#w1
   // the same network as SCL:
   #sRoofLeftDoorClosed(ACK := "F-DB_DataToSafety".ResetEmergencyStop AND #sAck_iRoofLeftDoorClosed,   // EV1oo2DI
                        IN1 := "FDI_RoofLeftDoorClosedCh1",
                        IN2 := "FDI_RoofLeftDoorClosedCh2",
                        DISCTIME := T#50MS,
                        Q => "F-DB_DataFromSafety".iRoofLeftDoorClosed,
                        ACK_REQ => #sAck_iRoofLeftDoorClosed);
END_REGION

REGION Network 12: Key Laser On
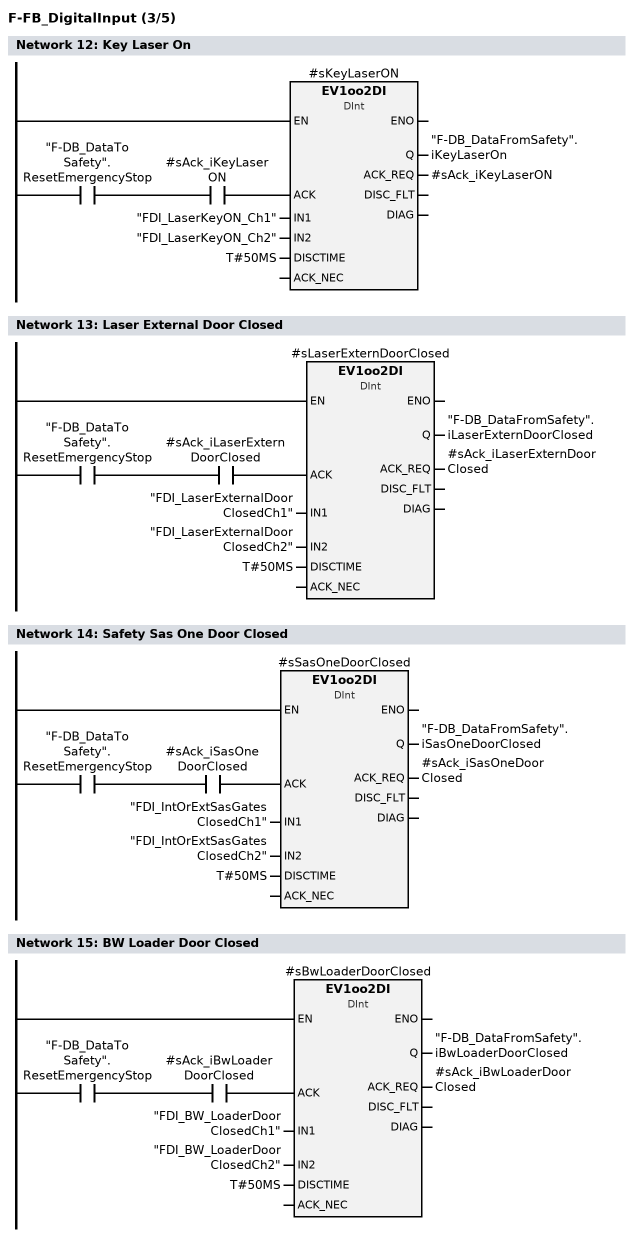
   RUNG wire#powerrail
      { S7_Templates := "codedbool_type := DInt" } #sKeyLaserON.EV1oo2DI(ACK := wire#w1, IN1 := "FDI_LaserKeyON_Ch1", IN2 := "FDI_LaserKeyON_Ch2", DISCTIME := T#50MS, ACK_NEC :=, Q => "F-DB_DataFromSafety".iKeyLaserOn, ACK_REQ => #sAck_iKeyLaserON, DISC_FLT =>, DIAG =>)
   END_RUNG
   RUNG wire#powerrail
      Contact( "F-DB_DataToSafety".ResetEmergencyStop )
      Contact( #sAck_iKeyLaserON )
   END_RUNG wire#w1
   // the same network as SCL:
   #sKeyLaserON(ACK := "F-DB_DataToSafety".ResetEmergencyStop AND #sAck_iKeyLaserON,   // EV1oo2DI
                IN1 := "FDI_LaserKeyON_Ch1",
                IN2 := "FDI_LaserKeyON_Ch2",
                DISCTIME := T#50MS,
                Q => "F-DB_DataFromSafety".iKeyLaserOn,
                ACK_REQ => #sAck_iKeyLaserON);
END_REGION

REGION Network 13: Laser External Door Closed
   RUNG wire#powerrail
      { S7_Templates := "codedbool_type := DInt" } #sLaserExternDoorClosed.EV1oo2DI(ACK := wire#w1, IN1 := "FDI_LaserExternalDoorClosedCh1", IN2 := "FDI_LaserExternalDoorClosedCh2", DISCTIME := T#50MS, ACK_NEC :=, Q => "F-DB_DataFromSafety".iLaserExternDoorClosed, ACK_REQ => #sAck_iLaserExternDoorClosed, DISC_FLT =>, DIAG =>)
   END_RUNG
   RUNG wire#powerrail
      Contact( "F-DB_DataToSafety".ResetEmergencyStop )
      Contact( #sAck_iLaserExternDoorClosed )
   END_RUNG wire#w1
   // the same network as SCL:
   #sLaserExternDoorClosed(ACK := "F-DB_DataToSafety".ResetEmergencyStop AND #sAck_iLaserExternDoorClosed,   // EV1oo2DI
                           IN1 := "FDI_LaserExternalDoorClosedCh1",
                           IN2 := "FDI_LaserExternalDoorClosedCh2",
                           DISCTIME := T#50MS,
                           Q => "F-DB_DataFromSafety".iLaserExternDoorClosed,
                           ACK_REQ => #sAck_iLaserExternDoorClosed);
END_REGION

REGION Network 14: Safety Sas One Door Closed
   RUNG wire#powerrail
      { S7_Templates := "codedbool_type := DInt" } #sSasOneDoorClosed.EV1oo2DI(ACK := wire#w1, IN1 := "FDI_IntOrExtSasGatesClosedCh1", IN2 := "FDI_IntOrExtSasGatesClosedCh2", DISCTIME := T#50MS, ACK_NEC :=, Q => "F-DB_DataFromSafety".iSasOneDoorClosed, ACK_REQ => #sAck_iSasOneDoorClosed, DISC_FLT =>, DIAG =>)
   END_RUNG
   RUNG wire#powerrail
      Contact( "F-DB_DataToSafety".ResetEmergencyStop )
      Contact( #sAck_iSasOneDoorClosed )
   END_RUNG wire#w1
   // the same network as SCL:
   #sSasOneDoorClosed(ACK := "F-DB_DataToSafety".ResetEmergencyStop AND #sAck_iSasOneDoorClosed,   // EV1oo2DI
                      IN1 := "FDI_IntOrExtSasGatesClosedCh1",
                      IN2 := "FDI_IntOrExtSasGatesClosedCh2",
                      DISCTIME := T#50MS,
                      Q => "F-DB_DataFromSafety".iSasOneDoorClosed,
                      ACK_REQ => #sAck_iSasOneDoorClosed);
END_REGION

REGION Network 15: BW Loader Door Closed
   RUNG wire#powerrail
      { S7_Templates := "codedbool_type := DInt" } #sBwLoaderDoorClosed.EV1oo2DI(ACK := wire#w1, IN1 := "FDI_BW_LoaderDoorClosedCh1", IN2 := "FDI_BW_LoaderDoorClosedCh2", DISCTIME := T#50MS, ACK_NEC :=, Q => "F-DB_DataFromSafety".iBwLoaderDoorClosed, ACK_REQ => #sAck_iBwLoaderDoorClosed, DISC_FLT =>, DIAG =>)
   END_RUNG
   RUNG wire#powerrail
      Contact( "F-DB_DataToSafety".ResetEmergencyStop )
      Contact( #sAck_iBwLoaderDoorClosed )
   END_RUNG wire#w1
   // the same network as SCL:
   #sBwLoaderDoorClosed(ACK := "F-DB_DataToSafety".ResetEmergencyStop AND #sAck_iBwLoaderDoorClosed,   // EV1oo2DI
                        IN1 := "FDI_BW_LoaderDoorClosedCh1",
                        IN2 := "FDI_BW_LoaderDoorClosedCh2",
                        DISCTIME := T#50MS,
                        Q => "F-DB_DataFromSafety".iBwLoaderDoorClosed,
                        ACK_REQ => #sAck_iBwLoaderDoorClosed);
END_REGION

REGION Network 16: Safety Right Door Closed
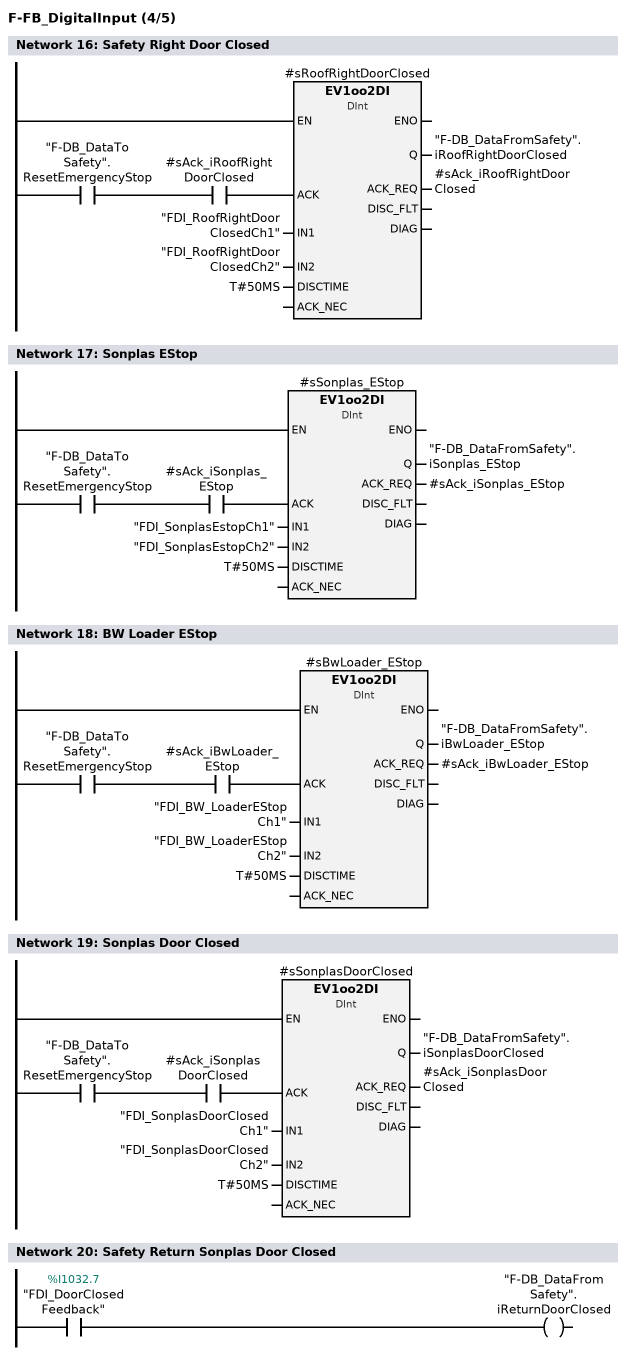
   RUNG wire#powerrail
      { S7_Templates := "codedbool_type := DInt" } #sRoofRightDoorClosed.EV1oo2DI(ACK := wire#w1, IN1 := "FDI_RoofRightDoorClosedCh1", IN2 := "FDI_RoofRightDoorClosedCh2", DISCTIME := T#50MS, ACK_NEC :=, Q => "F-DB_DataFromSafety".iRoofRightDoorClosed, ACK_REQ => #sAck_iRoofRightDoorClosed, DISC_FLT =>, DIAG =>)
   END_RUNG
   RUNG wire#powerrail
      Contact( "F-DB_DataToSafety".ResetEmergencyStop )
      Contact( #sAck_iRoofRightDoorClosed )
   END_RUNG wire#w1
   // the same network as SCL:
   #sRoofRightDoorClosed(ACK := "F-DB_DataToSafety".ResetEmergencyStop AND #sAck_iRoofRightDoorClosed,   // EV1oo2DI
                         IN1 := "FDI_RoofRightDoorClosedCh1",
                         IN2 := "FDI_RoofRightDoorClosedCh2",
                         DISCTIME := T#50MS,
                         Q => "F-DB_DataFromSafety".iRoofRightDoorClosed,
                         ACK_REQ => #sAck_iRoofRightDoorClosed);
END_REGION

REGION Network 17: Sonplas EStop
   RUNG wire#powerrail
      { S7_Templates := "codedbool_type := DInt" } #sSonplas_EStop.EV1oo2DI(ACK := wire#w1, IN1 := "FDI_SonplasEstopCh1", IN2 := "FDI_SonplasEstopCh2", DISCTIME := T#50MS, ACK_NEC :=, Q => "F-DB_DataFromSafety".iSonplas_EStop, ACK_REQ => #sAck_iSonplas_EStop, DISC_FLT =>, DIAG =>)
   END_RUNG
   RUNG wire#powerrail
      Contact( "F-DB_DataToSafety".ResetEmergencyStop )
      Contact( #sAck_iSonplas_EStop )
   END_RUNG wire#w1
   // the same network as SCL:
   #sSonplas_EStop(ACK := "F-DB_DataToSafety".ResetEmergencyStop AND #sAck_iSonplas_EStop,   // EV1oo2DI
                   IN1 := "FDI_SonplasEstopCh1",
                   IN2 := "FDI_SonplasEstopCh2",
                   DISCTIME := T#50MS,
                   Q => "F-DB_DataFromSafety".iSonplas_EStop,
                   ACK_REQ => #sAck_iSonplas_EStop);
END_REGION

REGION Network 18: BW Loader EStop
   RUNG wire#powerrail
      { S7_Templates := "codedbool_type := DInt" } #sBwLoader_EStop.EV1oo2DI(ACK := wire#w1, IN1 := "FDI_BW_LoaderEStopCh1", IN2 := "FDI_BW_LoaderEStopCh2", DISCTIME := T#50MS, ACK_NEC :=, Q => "F-DB_DataFromSafety".iBwLoader_EStop, ACK_REQ => #sAck_iBwLoader_EStop, DISC_FLT =>, DIAG =>)
   END_RUNG
   RUNG wire#powerrail
      Contact( "F-DB_DataToSafety".ResetEmergencyStop )
      Contact( #sAck_iBwLoader_EStop )
   END_RUNG wire#w1
   // the same network as SCL:
   #sBwLoader_EStop(ACK := "F-DB_DataToSafety".ResetEmergencyStop AND #sAck_iBwLoader_EStop,   // EV1oo2DI
                    IN1 := "FDI_BW_LoaderEStopCh1",
                    IN2 := "FDI_BW_LoaderEStopCh2",
                    DISCTIME := T#50MS,
                    Q => "F-DB_DataFromSafety".iBwLoader_EStop,
                    ACK_REQ => #sAck_iBwLoader_EStop);
END_REGION

REGION Network 19: Sonplas Door Closed
   RUNG wire#powerrail
      { S7_Templates := "codedbool_type := DInt" } #sSonplasDoorClosed.EV1oo2DI(ACK := wire#w1, IN1 := "FDI_SonplasDoorClosedCh1", IN2 := "FDI_SonplasDoorClosedCh2", DISCTIME := T#50MS, ACK_NEC :=, Q => "F-DB_DataFromSafety".iSonplasDoorClosed, ACK_REQ => #sAck_iSonplasDoorClosed, DISC_FLT =>, DIAG =>)
   END_RUNG
   RUNG wire#powerrail
      Contact( "F-DB_DataToSafety".ResetEmergencyStop )
      Contact( #sAck_iSonplasDoorClosed )
   END_RUNG wire#w1
   // the same network as SCL:
   #sSonplasDoorClosed(ACK := "F-DB_DataToSafety".ResetEmergencyStop AND #sAck_iSonplasDoorClosed,   // EV1oo2DI
                       IN1 := "FDI_SonplasDoorClosedCh1",
                       IN2 := "FDI_SonplasDoorClosedCh2",
                       DISCTIME := T#50MS,
                       Q => "F-DB_DataFromSafety".iSonplasDoorClosed,
                       ACK_REQ => #sAck_iSonplasDoorClosed);
END_REGION

REGION Network 20: Safety Return Sonplas Door Closed
   RUNG wire#powerrail
      Contact( "FDI_DoorClosedFeedback" )
      Coil( "F-DB_DataFromSafety".iReturnDoorClosed )
   END_RUNG
   // the same network as SCL:
   "F-DB_DataFromSafety".iReturnDoorClosed := "FDI_DoorClosedFeedback";
END_REGION

REGION Network 21: Manage Acknowledge Request
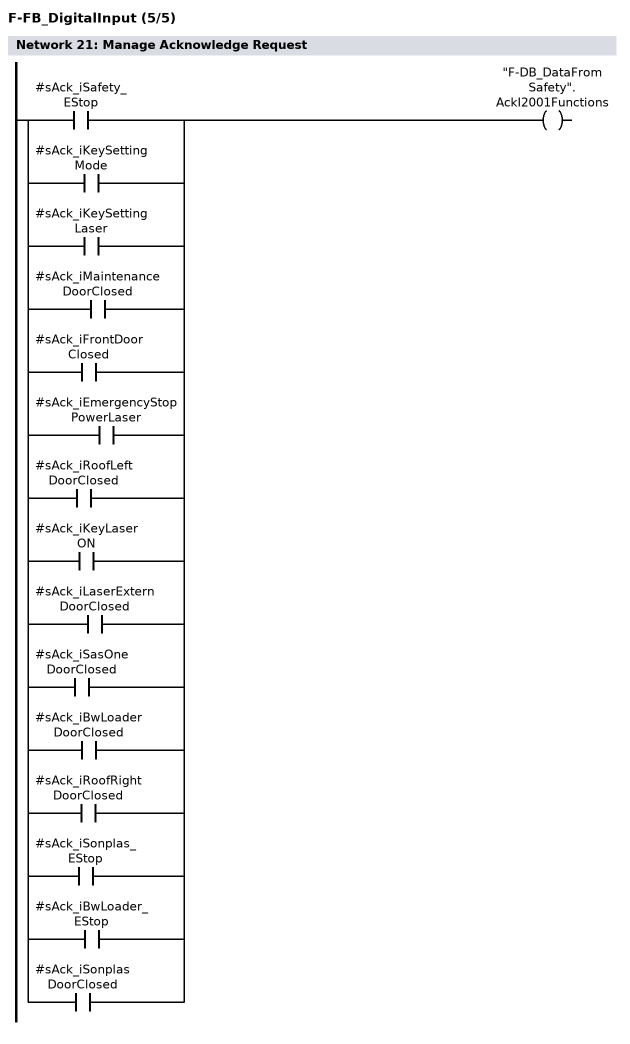
   RUNG wire#powerrail
      Contact( #sAck_iSafety_EStop )
      wire#w1
      Coil( "F-DB_DataFromSafety".AckI2001Functions )
   END_RUNG
   RUNG wire#powerrail
      Contact( #sAck_iKeySettingMode )
   END_RUNG wire#w1
   RUNG wire#powerrail
      Contact( #sAck_iKeySettingLaser )
   END_RUNG wire#w1
   RUNG wire#powerrail
      Contact( #sAck_iMaintenanceDoorClosed )
   END_RUNG wire#w1
   RUNG wire#powerrail
      Contact( #sAck_iFrontDoorClosed )
   END_RUNG wire#w1
   RUNG wire#powerrail
      Contact( #sAck_iEmergencyStopPowerLaser )
   END_RUNG wire#w1
   RUNG wire#powerrail
      Contact( #sAck_iRoofLeftDoorClosed )
   END_RUNG wire#w1
   RUNG wire#powerrail
      Contact( #sAck_iKeyLaserON )
   END_RUNG wire#w1
   RUNG wire#powerrail
      Contact( #sAck_iLaserExternDoorClosed )
   END_RUNG wire#w1
   RUNG wire#powerrail
      Contact( #sAck_iSasOneDoorClosed )
   END_RUNG wire#w1
   RUNG wire#powerrail
      Contact( #sAck_iBwLoaderDoorClosed )
   END_RUNG wire#w1
   RUNG wire#powerrail
      Contact( #sAck_iRoofRightDoorClosed )
   END_RUNG wire#w1
   RUNG wire#powerrail
      Contact( #sAck_iSonplas_EStop )
   END_RUNG wire#w1
   RUNG wire#powerrail
      Contact( #sAck_iBwLoader_EStop )
   END_RUNG wire#w1
   RUNG wire#powerrail
      Contact( #sAck_iSonplasDoorClosed )
   END_RUNG wire#w1
   // the same network as SCL:
   "F-DB_DataFromSafety".AckI2001Functions := #sAck_iSafety_EStop OR #sAck_iKeySettingMode OR #sAck_iKeySettingLaser OR #sAck_iMaintenanceDoorClosed OR #sAck_iFrontDoorClosed OR #sAck_iEmergencyStopPowerLaser OR #sAck_iRoofLeftDoorClosed OR #sAck_iKeyLaserON OR #sAck_iLaserExternDoorClosed OR #sAck_iSasOneDoorClosed OR #sAck_iBwLoaderDoorClosed OR #sAck_iRoofRightDoorClosed OR #sAck_iSonplas_EStop OR #sAck_iBwLoader_EStop OR #sAck_iSonplasDoorClosed;
END_REGION
END_FUNCTION_BLOCK

FUNCTION_BLOCK "F-FB_Axis"   // FB130, F_LAD
{ S7_Optimized_Access := 'TRUE' }
// stored: AutoNumber false
   VAR
      LDrvSafe_SinaTlg903StatusAxis01_X : "LDrvSafe_SinaTlg903Status";
      LDrvSafe_SinaTlg903StatusAxis02_Y : "LDrvSafe_SinaTlg903Status";
      LDrvSafe_SinaTlg903StatusAxis03_ZM : "LDrvSafe_SinaTlg903Status";
      LDrvSafe_SinaTlg903StatusAxis04_B : "LDrvSafe_SinaTlg903Status";
      LDrvSafe_SinaTlg903StatusAxis05_U1 : "LDrvSafe_SinaTlg903Status";
      LDrvSafe_SinaTlg903StatusAxis06_U2 : "LDrvSafe_SinaTlg903Status";
      LDrvSafe_SinaTlg903StatusAxis07_V : "LDrvSafe_SinaTlg903Status";
      LDrvSafe_SinaTlg903StatusAxis08_W : "LDrvSafe_SinaTlg903Status";
      LDrvSafe_SinaTlg903StatusAxis09_ZL : "LDrvSafe_SinaTlg903Status";
      LDrvSafe_SinaTlg903ControlAxis01_X : "LDrvSafe_SinaTlg903Control";
      LDrvSafe_SinaTlg903ControlAxis02_Y : "LDrvSafe_SinaTlg903Control";
      LDrvSafe_SinaTlg903ControlAxis03_ZM : "LDrvSafe_SinaTlg903Control";
      LDrvSafe_SinaTlg903ControlAxis04_B : "LDrvSafe_SinaTlg903Control";
      LDrvSafe_SinaTlg903ControlAxis05_U1 : "LDrvSafe_SinaTlg903Control";
      LDrvSafe_SinaTlg903ControlAxis06_U2 : "LDrvSafe_SinaTlg903Control";
      LDrvSafe_SinaTlg903ControlAxis07_V : "LDrvSafe_SinaTlg903Control";
      LDrvSafe_SinaTlg903ControlAxis08_W : "LDrvSafe_SinaTlg903Control";
      LDrvSafe_SinaTlg903ControlAxis09_ZL : "LDrvSafe_SinaTlg903Control";
   END_VAR
   VAR_TEMP
      tEnable_Axis_Move : Bool;
   END_VAR
BEGIN

REGION Network 1: Enable Axis Move
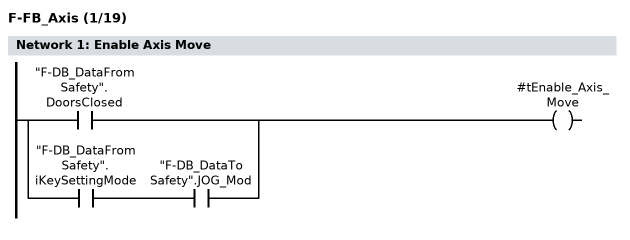
   RUNG wire#powerrail
      Contact( "F-DB_DataFromSafety".DoorsClosed )
      wire#w1
      Coil( #tEnable_Axis_Move )
   END_RUNG
   RUNG wire#powerrail
      Contact( "F-DB_DataFromSafety".iKeySettingMode )
      Contact( "F-DB_DataToSafety".JOG_Mod )
   END_RUNG wire#w1
   // the same network as SCL:
   #tEnable_Axis_Move := "F-DB_DataFromSafety".DoorsClosed OR ("F-DB_DataFromSafety".iKeySettingMode AND "F-DB_DataToSafety".JOG_Mod);
END_REGION

REGION Network 2: Axis01_X Status
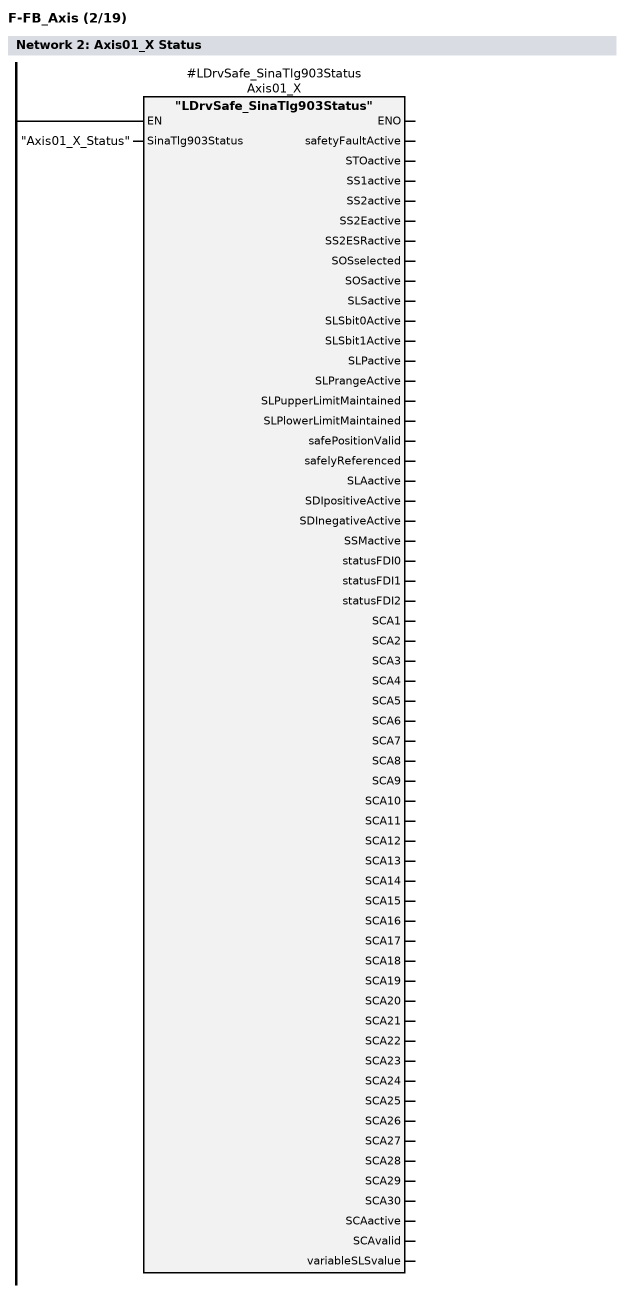
   RUNG wire#powerrail
      #LDrvSafe_SinaTlg903StatusAxis01_X(SinaTlg903Status := "Axis01_X_Status", safetyFaultActive =>, STOactive =>, SS1active =>, SS2active =>, SS2Eactive =>, SS2ESRactive =>, SOSselected =>, SOSactive =>, SLSactive =>, SLSbit0Active =>, SLSbit1Active =>, SLPactive =>, SLPrangeActive =>, SLPupperLimitMaintained =>, SLPlowerLimitMaintained =>, safePositionValid =>, safelyReferenced =>, SLAactive =>, SDIpositiveActive =>, SDInegativeActive =>, SSMactive =>, statusFDI0 =>, statusFDI1 =>, statusFDI2 =>, SCA1 =>, SCA2 =>, SCA3 =>, SCA4 =>, SCA5 =>, SCA6 =>, SCA7 =>, SCA8 =>, SCA9 =>, SCA10 =>, SCA11 =>, SCA12 =>, SCA13 =>, SCA14 =>, SCA15 =>, SCA16 =>, SCA17 =>, SCA18 =>, SCA19 =>, SCA20 =>, SCA21 =>, SCA22 =>, SCA23 =>, SCA24 =>, SCA25 =>, SCA26 =>, SCA27 =>, SCA28 =>, SCA29 =>, SCA30 =>, SCAactive =>, SCAvalid =>, variableSLSvalue =>)
   END_RUNG
   // the same network as SCL:
   #LDrvSafe_SinaTlg903StatusAxis01_X(SinaTlg903Status := "Axis01_X_Status");   // "LDrvSafe_SinaTlg903Status"
END_REGION

REGION Network 3: Axis01_X Control
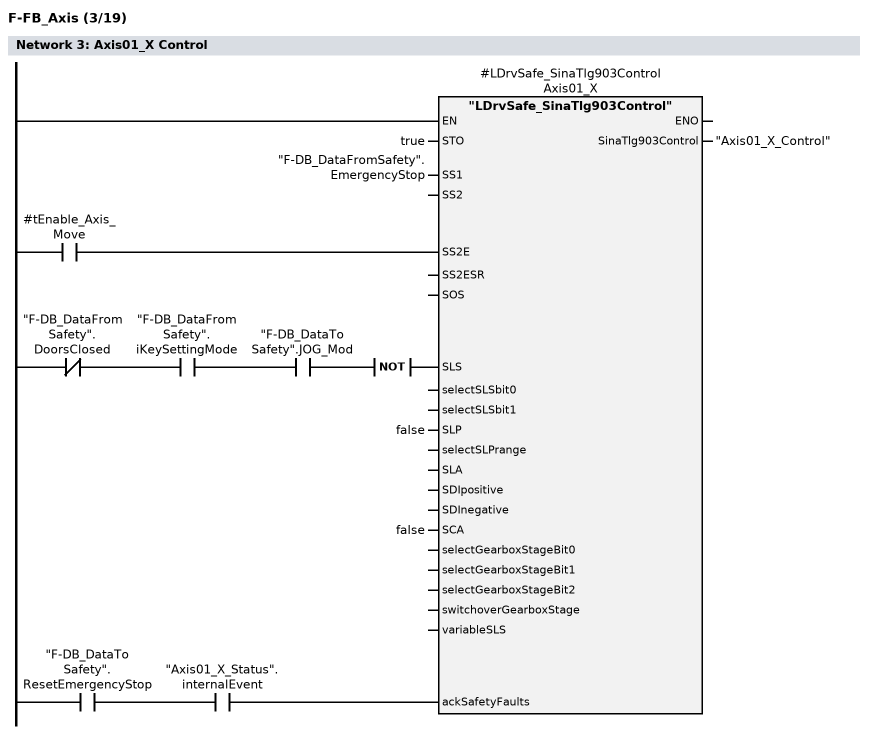
   RUNG wire#powerrail
      #LDrvSafe_SinaTlg903ControlAxis01_X(SS2E := wire#w1, SLS := wire#w2, ackSafetyFaults := wire#w3, STO := true, SS1 := "F-DB_DataFromSafety".EmergencyStop, SS2 :=, SS2ESR :=, SOS :=, selectSLSbit0 :=, selectSLSbit1 :=, SLP := false, selectSLPrange :=, SLA :=, SDIpositive :=, SDInegative :=, SCA := false, selectGearboxStageBit0 :=, selectGearboxStageBit1 :=, selectGearboxStageBit2 :=, switchoverGearboxStage :=, variableSLS :=, SinaTlg903Control => "Axis01_X_Control")
   END_RUNG
   RUNG wire#powerrail
      Contact( #tEnable_Axis_Move )
   END_RUNG wire#w1
   RUNG wire#powerrail
      I_Contact( "F-DB_DataFromSafety".DoorsClosed )
      Contact( "F-DB_DataFromSafety".iKeySettingMode )
      Contact( "F-DB_DataToSafety".JOG_Mod )
      Not()
   END_RUNG wire#w2
   RUNG wire#powerrail
      Contact( "F-DB_DataToSafety".ResetEmergencyStop )
      Contact( "Axis01_X_Status".internalEvent )
   END_RUNG wire#w3
   // the same network as SCL:
   #LDrvSafe_SinaTlg903ControlAxis01_X(STO := true,   // "LDrvSafe_SinaTlg903Control"
                           SS1 := "F-DB_DataFromSafety".EmergencyStop,
                           SS2E := #tEnable_Axis_Move,
                           SLS := NOT (NOT "F-DB_DataFromSafety".DoorsClosed AND "F-DB_DataFromSafety".iKeySettingMode AND "F-DB_DataToSafety".JOG_Mod),
                           SLP := false,
                           SCA := false,
                           ackSafetyFaults := "F-DB_DataToSafety".ResetEmergencyStop AND "Axis01_X_Status".internalEvent,
                           SinaTlg903Control => "Axis01_X_Control");
END_REGION

REGION Network 4: Axis02_Y Status
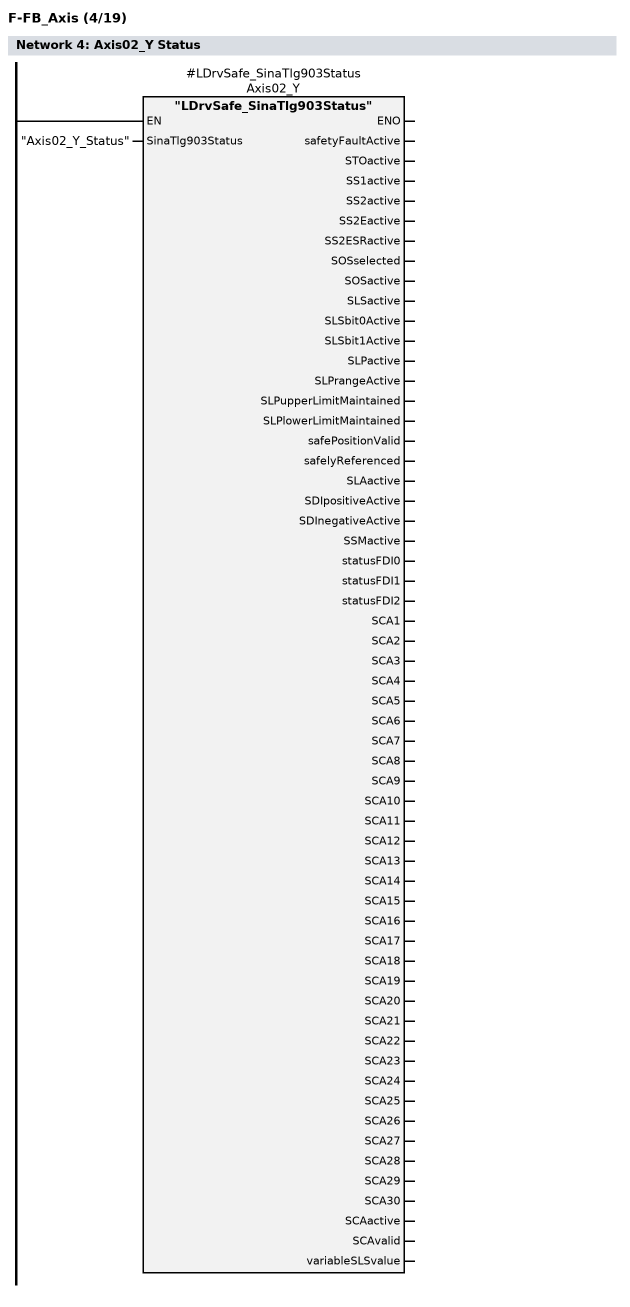
   RUNG wire#powerrail
      #LDrvSafe_SinaTlg903StatusAxis02_Y(SinaTlg903Status := "Axis02_Y_Status", safetyFaultActive =>, STOactive =>, SS1active =>, SS2active =>, SS2Eactive =>, SS2ESRactive =>, SOSselected =>, SOSactive =>, SLSactive =>, SLSbit0Active =>, SLSbit1Active =>, SLPactive =>, SLPrangeActive =>, SLPupperLimitMaintained =>, SLPlowerLimitMaintained =>, safePositionValid =>, safelyReferenced =>, SLAactive =>, SDIpositiveActive =>, SDInegativeActive =>, SSMactive =>, statusFDI0 =>, statusFDI1 =>, statusFDI2 =>, SCA1 =>, SCA2 =>, SCA3 =>, SCA4 =>, SCA5 =>, SCA6 =>, SCA7 =>, SCA8 =>, SCA9 =>, SCA10 =>, SCA11 =>, SCA12 =>, SCA13 =>, SCA14 =>, SCA15 =>, SCA16 =>, SCA17 =>, SCA18 =>, SCA19 =>, SCA20 =>, SCA21 =>, SCA22 =>, SCA23 =>, SCA24 =>, SCA25 =>, SCA26 =>, SCA27 =>, SCA28 =>, SCA29 =>, SCA30 =>, SCAactive =>, SCAvalid =>, variableSLSvalue =>)
   END_RUNG
   // the same network as SCL:
   #LDrvSafe_SinaTlg903StatusAxis02_Y(SinaTlg903Status := "Axis02_Y_Status");   // "LDrvSafe_SinaTlg903Status"
END_REGION

REGION Network 5: Axis02_Y Control
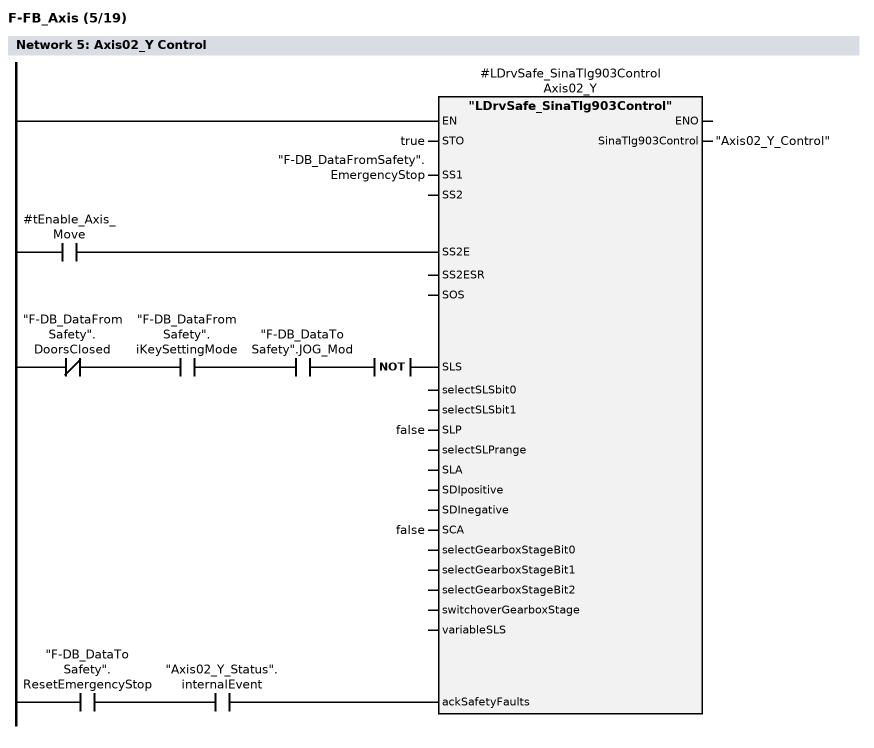
   RUNG wire#powerrail
      #LDrvSafe_SinaTlg903ControlAxis02_Y(SS2E := wire#w1, SLS := wire#w2, ackSafetyFaults := wire#w3, STO := true, SS1 := "F-DB_DataFromSafety".EmergencyStop, SS2 :=, SS2ESR :=, SOS :=, selectSLSbit0 :=, selectSLSbit1 :=, SLP := false, selectSLPrange :=, SLA :=, SDIpositive :=, SDInegative :=, SCA := false, selectGearboxStageBit0 :=, selectGearboxStageBit1 :=, selectGearboxStageBit2 :=, switchoverGearboxStage :=, variableSLS :=, SinaTlg903Control => "Axis02_Y_Control")
   END_RUNG
   RUNG wire#powerrail
      Contact( #tEnable_Axis_Move )
   END_RUNG wire#w1
   RUNG wire#powerrail
      I_Contact( "F-DB_DataFromSafety".DoorsClosed )
      Contact( "F-DB_DataFromSafety".iKeySettingMode )
      Contact( "F-DB_DataToSafety".JOG_Mod )
      Not()
   END_RUNG wire#w2
   RUNG wire#powerrail
      Contact( "F-DB_DataToSafety".ResetEmergencyStop )
      Contact( "Axis02_Y_Status".internalEvent )
   END_RUNG wire#w3
   // the same network as SCL:
   #LDrvSafe_SinaTlg903ControlAxis02_Y(STO := true,   // "LDrvSafe_SinaTlg903Control"
                           SS1 := "F-DB_DataFromSafety".EmergencyStop,
                           SS2E := #tEnable_Axis_Move,
                           SLS := NOT (NOT "F-DB_DataFromSafety".DoorsClosed AND "F-DB_DataFromSafety".iKeySettingMode AND "F-DB_DataToSafety".JOG_Mod),
                           SLP := false,
                           SCA := false,
                           ackSafetyFaults := "F-DB_DataToSafety".ResetEmergencyStop AND "Axis02_Y_Status".internalEvent,
                           SinaTlg903Control => "Axis02_Y_Control");
END_REGION

REGION Network 6: Axis03_ZM Status
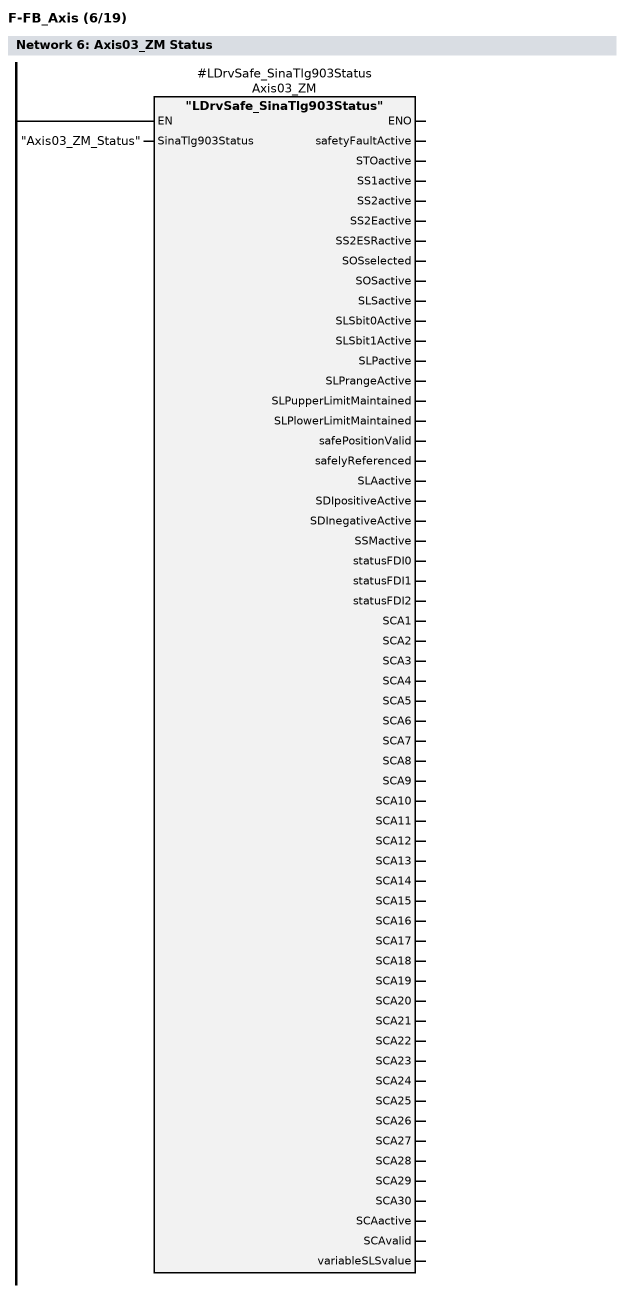
   RUNG wire#powerrail
      #LDrvSafe_SinaTlg903StatusAxis03_ZM(SinaTlg903Status := "Axis03_ZM_Status", safetyFaultActive =>, STOactive =>, SS1active =>, SS2active =>, SS2Eactive =>, SS2ESRactive =>, SOSselected =>, SOSactive =>, SLSactive =>, SLSbit0Active =>, SLSbit1Active =>, SLPactive =>, SLPrangeActive =>, SLPupperLimitMaintained =>, SLPlowerLimitMaintained =>, safePositionValid =>, safelyReferenced =>, SLAactive =>, SDIpositiveActive =>, SDInegativeActive =>, SSMactive =>, statusFDI0 =>, statusFDI1 =>, statusFDI2 =>, SCA1 =>, SCA2 =>, SCA3 =>, SCA4 =>, SCA5 =>, SCA6 =>, SCA7 =>, SCA8 =>, SCA9 =>, SCA10 =>, SCA11 =>, SCA12 =>, SCA13 =>, SCA14 =>, SCA15 =>, SCA16 =>, SCA17 =>, SCA18 =>, SCA19 =>, SCA20 =>, SCA21 =>, SCA22 =>, SCA23 =>, SCA24 =>, SCA25 =>, SCA26 =>, SCA27 =>, SCA28 =>, SCA29 =>, SCA30 =>, SCAactive =>, SCAvalid =>, variableSLSvalue =>)
   END_RUNG
   // the same network as SCL:
   #LDrvSafe_SinaTlg903StatusAxis03_ZM(SinaTlg903Status := "Axis03_ZM_Status");   // "LDrvSafe_SinaTlg903Status"
END_REGION

REGION Network 7: Axis03_ZM Control
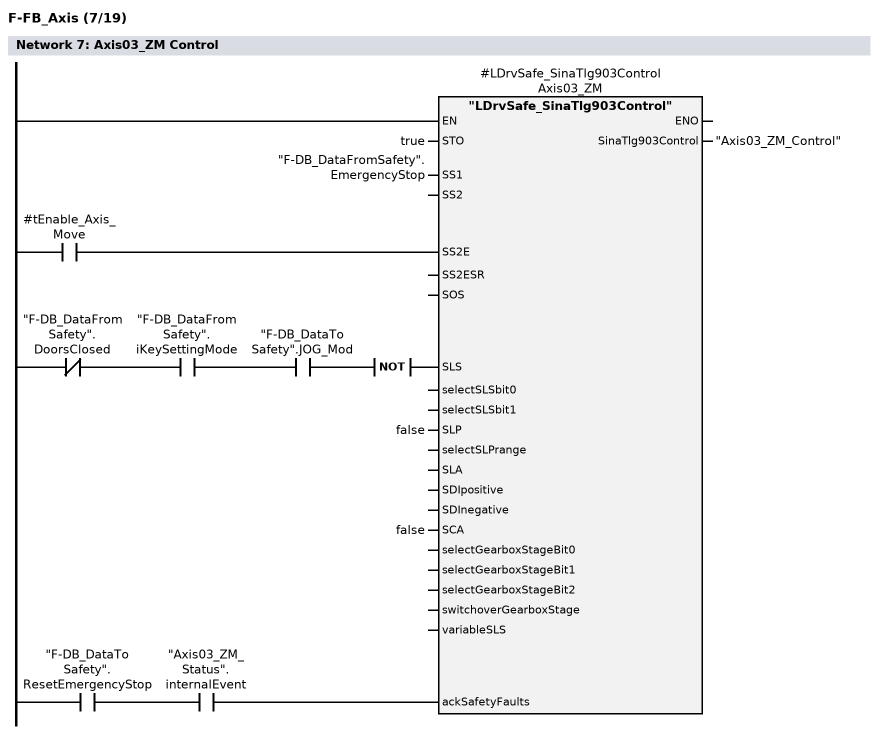
   RUNG wire#powerrail
      #LDrvSafe_SinaTlg903ControlAxis03_ZM(SS2E := wire#w1, SLS := wire#w2, ackSafetyFaults := wire#w3, STO := true, SS1 := "F-DB_DataFromSafety".EmergencyStop, SS2 :=, SS2ESR :=, SOS :=, selectSLSbit0 :=, selectSLSbit1 :=, SLP := false, selectSLPrange :=, SLA :=, SDIpositive :=, SDInegative :=, SCA := false, selectGearboxStageBit0 :=, selectGearboxStageBit1 :=, selectGearboxStageBit2 :=, switchoverGearboxStage :=, variableSLS :=, SinaTlg903Control => "Axis03_ZM_Control")
   END_RUNG
   RUNG wire#powerrail
      Contact( #tEnable_Axis_Move )
   END_RUNG wire#w1
   RUNG wire#powerrail
      I_Contact( "F-DB_DataFromSafety".DoorsClosed )
      Contact( "F-DB_DataFromSafety".iKeySettingMode )
      Contact( "F-DB_DataToSafety".JOG_Mod )
      Not()
   END_RUNG wire#w2
   RUNG wire#powerrail
      Contact( "F-DB_DataToSafety".ResetEmergencyStop )
      Contact( "Axis03_ZM_Status".internalEvent )
   END_RUNG wire#w3
   // the same network as SCL:
   #LDrvSafe_SinaTlg903ControlAxis03_ZM(STO := true,   // "LDrvSafe_SinaTlg903Control"
                           SS1 := "F-DB_DataFromSafety".EmergencyStop,
                           SS2E := #tEnable_Axis_Move,
                           SLS := NOT (NOT "F-DB_DataFromSafety".DoorsClosed AND "F-DB_DataFromSafety".iKeySettingMode AND "F-DB_DataToSafety".JOG_Mod),
                           SLP := false,
                           SCA := false,
                           ackSafetyFaults := "F-DB_DataToSafety".ResetEmergencyStop AND "Axis03_ZM_Status".internalEvent,
                           SinaTlg903Control => "Axis03_ZM_Control");
END_REGION

REGION Network 8: Axis04_B Status
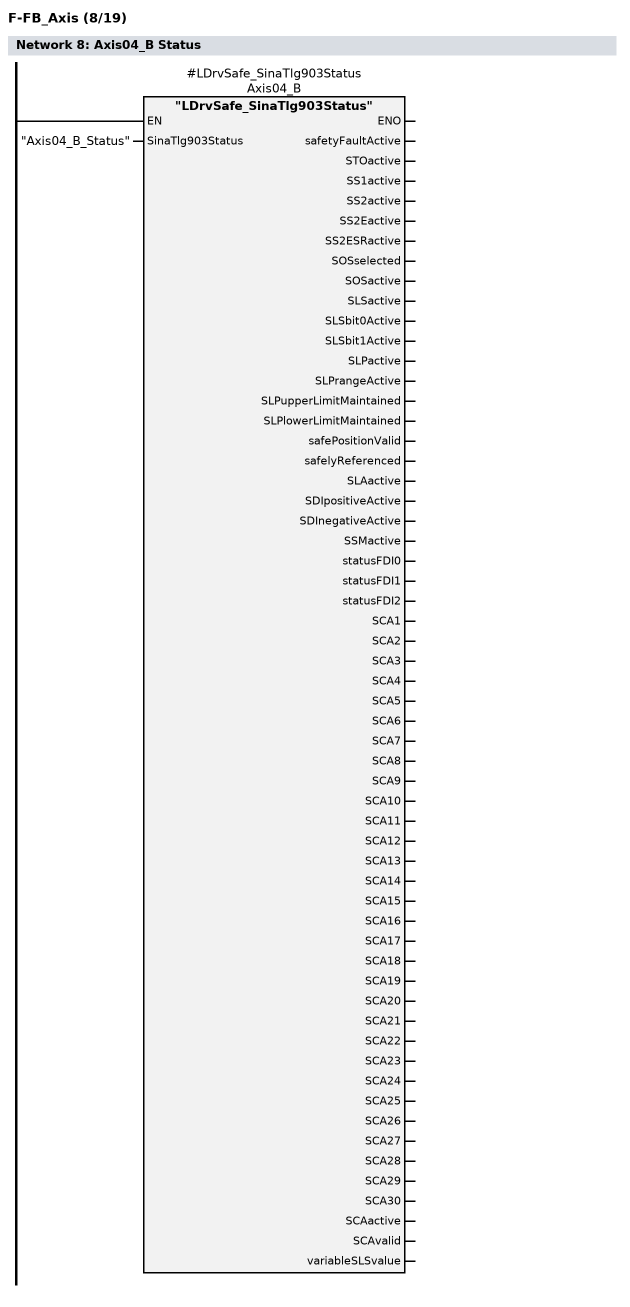
   RUNG wire#powerrail
      #LDrvSafe_SinaTlg903StatusAxis04_B(SinaTlg903Status := "Axis04_B_Status", safetyFaultActive =>, STOactive =>, SS1active =>, SS2active =>, SS2Eactive =>, SS2ESRactive =>, SOSselected =>, SOSactive =>, SLSactive =>, SLSbit0Active =>, SLSbit1Active =>, SLPactive =>, SLPrangeActive =>, SLPupperLimitMaintained =>, SLPlowerLimitMaintained =>, safePositionValid =>, safelyReferenced =>, SLAactive =>, SDIpositiveActive =>, SDInegativeActive =>, SSMactive =>, statusFDI0 =>, statusFDI1 =>, statusFDI2 =>, SCA1 =>, SCA2 =>, SCA3 =>, SCA4 =>, SCA5 =>, SCA6 =>, SCA7 =>, SCA8 =>, SCA9 =>, SCA10 =>, SCA11 =>, SCA12 =>, SCA13 =>, SCA14 =>, SCA15 =>, SCA16 =>, SCA17 =>, SCA18 =>, SCA19 =>, SCA20 =>, SCA21 =>, SCA22 =>, SCA23 =>, SCA24 =>, SCA25 =>, SCA26 =>, SCA27 =>, SCA28 =>, SCA29 =>, SCA30 =>, SCAactive =>, SCAvalid =>, variableSLSvalue =>)
   END_RUNG
   // the same network as SCL:
   #LDrvSafe_SinaTlg903StatusAxis04_B(SinaTlg903Status := "Axis04_B_Status");   // "LDrvSafe_SinaTlg903Status"
END_REGION

REGION Network 9: Axis04_B Control
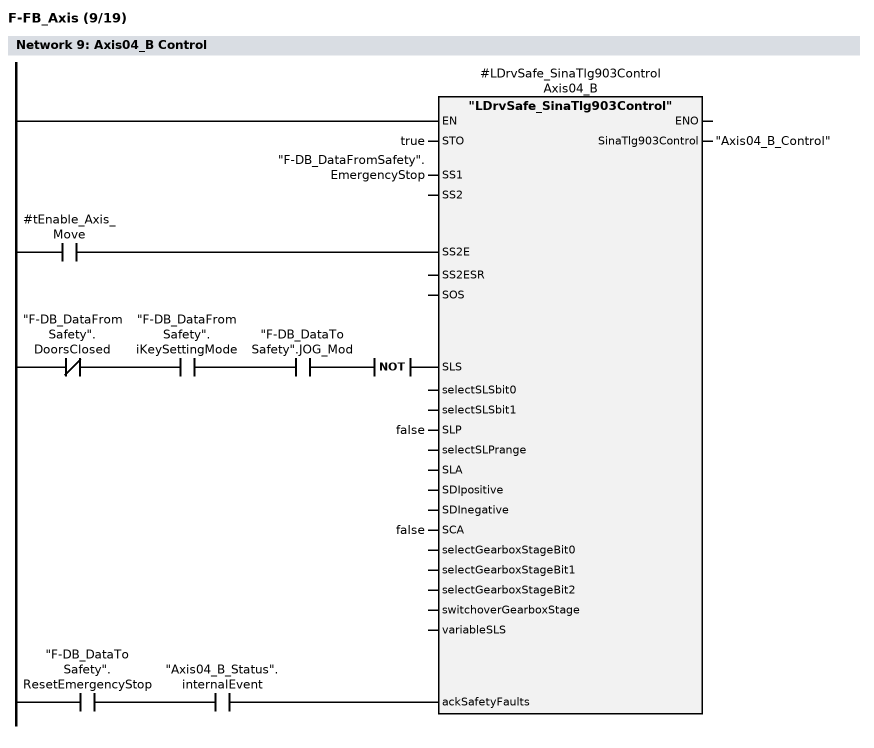
   RUNG wire#powerrail
      #LDrvSafe_SinaTlg903ControlAxis04_B(SS2E := wire#w1, SLS := wire#w2, ackSafetyFaults := wire#w3, STO := true, SS1 := "F-DB_DataFromSafety".EmergencyStop, SS2 :=, SS2ESR :=, SOS :=, selectSLSbit0 :=, selectSLSbit1 :=, SLP := false, selectSLPrange :=, SLA :=, SDIpositive :=, SDInegative :=, SCA := false, selectGearboxStageBit0 :=, selectGearboxStageBit1 :=, selectGearboxStageBit2 :=, switchoverGearboxStage :=, variableSLS :=, SinaTlg903Control => "Axis04_B_Control")
   END_RUNG
   RUNG wire#powerrail
      Contact( #tEnable_Axis_Move )
   END_RUNG wire#w1
   RUNG wire#powerrail
      I_Contact( "F-DB_DataFromSafety".DoorsClosed )
      Contact( "F-DB_DataFromSafety".iKeySettingMode )
      Contact( "F-DB_DataToSafety".JOG_Mod )
      Not()
   END_RUNG wire#w2
   RUNG wire#powerrail
      Contact( "F-DB_DataToSafety".ResetEmergencyStop )
      Contact( "Axis04_B_Status".internalEvent )
   END_RUNG wire#w3
   // the same network as SCL:
   #LDrvSafe_SinaTlg903ControlAxis04_B(STO := true,   // "LDrvSafe_SinaTlg903Control"
                           SS1 := "F-DB_DataFromSafety".EmergencyStop,
                           SS2E := #tEnable_Axis_Move,
                           SLS := NOT (NOT "F-DB_DataFromSafety".DoorsClosed AND "F-DB_DataFromSafety".iKeySettingMode AND "F-DB_DataToSafety".JOG_Mod),
                           SLP := false,
                           SCA := false,
                           ackSafetyFaults := "F-DB_DataToSafety".ResetEmergencyStop AND "Axis04_B_Status".internalEvent,
                           SinaTlg903Control => "Axis04_B_Control");
END_REGION

REGION Network 10: Axis05_U1 Status
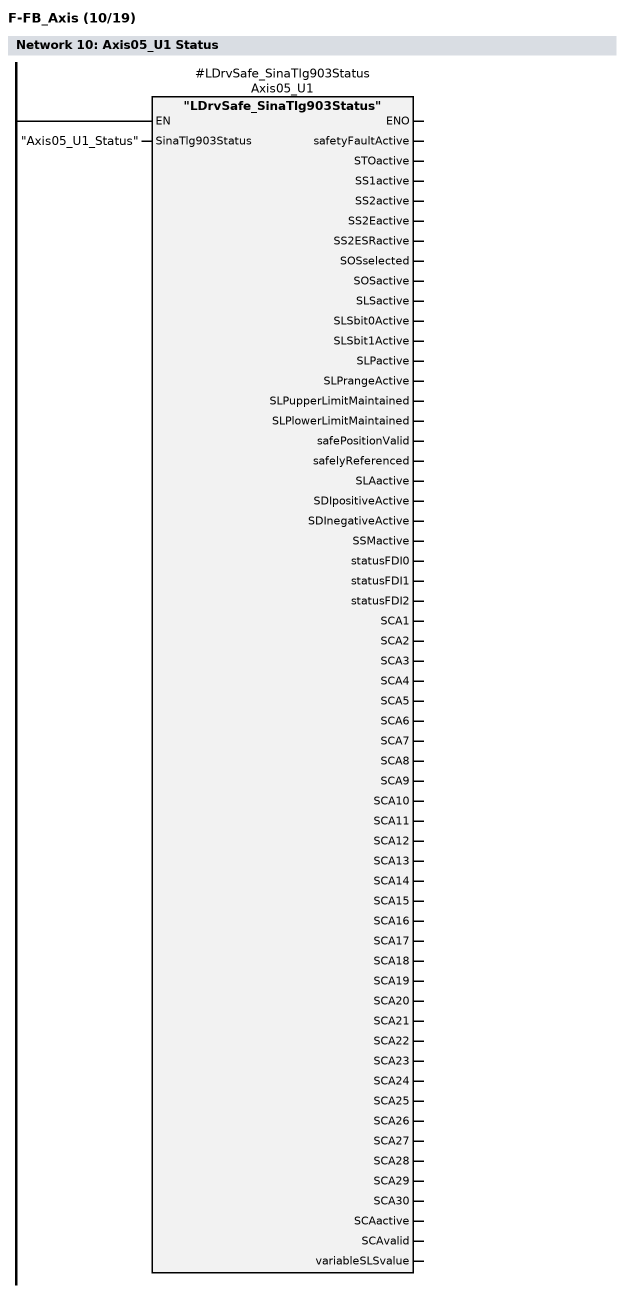
   RUNG wire#powerrail
      #LDrvSafe_SinaTlg903StatusAxis05_U1(SinaTlg903Status := "Axis05_U1_Status", safetyFaultActive =>, STOactive =>, SS1active =>, SS2active =>, SS2Eactive =>, SS2ESRactive =>, SOSselected =>, SOSactive =>, SLSactive =>, SLSbit0Active =>, SLSbit1Active =>, SLPactive =>, SLPrangeActive =>, SLPupperLimitMaintained =>, SLPlowerLimitMaintained =>, safePositionValid =>, safelyReferenced =>, SLAactive =>, SDIpositiveActive =>, SDInegativeActive =>, SSMactive =>, statusFDI0 =>, statusFDI1 =>, statusFDI2 =>, SCA1 =>, SCA2 =>, SCA3 =>, SCA4 =>, SCA5 =>, SCA6 =>, SCA7 =>, SCA8 =>, SCA9 =>, SCA10 =>, SCA11 =>, SCA12 =>, SCA13 =>, SCA14 =>, SCA15 =>, SCA16 =>, SCA17 =>, SCA18 =>, SCA19 =>, SCA20 =>, SCA21 =>, SCA22 =>, SCA23 =>, SCA24 =>, SCA25 =>, SCA26 =>, SCA27 =>, SCA28 =>, SCA29 =>, SCA30 =>, SCAactive =>, SCAvalid =>, variableSLSvalue =>)
   END_RUNG
   // the same network as SCL:
   #LDrvSafe_SinaTlg903StatusAxis05_U1(SinaTlg903Status := "Axis05_U1_Status");   // "LDrvSafe_SinaTlg903Status"
END_REGION

REGION Network 11: Axis05_U1 Control
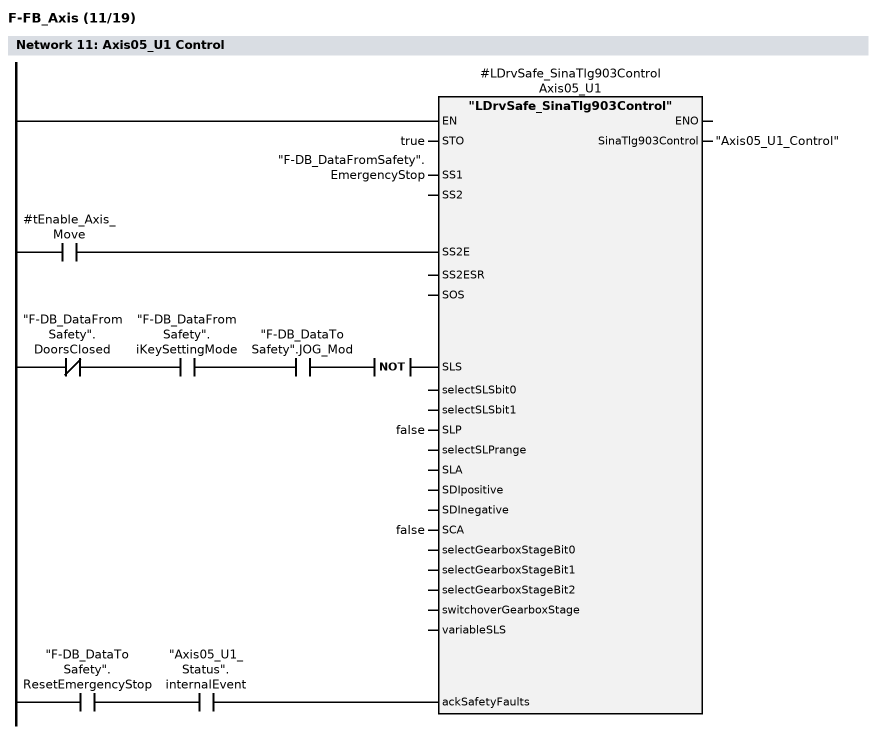
   RUNG wire#powerrail
      #LDrvSafe_SinaTlg903ControlAxis05_U1(SS2E := wire#w1, SLS := wire#w2, ackSafetyFaults := wire#w3, STO := true, SS1 := "F-DB_DataFromSafety".EmergencyStop, SS2 :=, SS2ESR :=, SOS :=, selectSLSbit0 :=, selectSLSbit1 :=, SLP := false, selectSLPrange :=, SLA :=, SDIpositive :=, SDInegative :=, SCA := false, selectGearboxStageBit0 :=, selectGearboxStageBit1 :=, selectGearboxStageBit2 :=, switchoverGearboxStage :=, variableSLS :=, SinaTlg903Control => "Axis05_U1_Control")
   END_RUNG
   RUNG wire#powerrail
      Contact( #tEnable_Axis_Move )
   END_RUNG wire#w1
   RUNG wire#powerrail
      I_Contact( "F-DB_DataFromSafety".DoorsClosed )
      Contact( "F-DB_DataFromSafety".iKeySettingMode )
      Contact( "F-DB_DataToSafety".JOG_Mod )
      Not()
   END_RUNG wire#w2
   RUNG wire#powerrail
      Contact( "F-DB_DataToSafety".ResetEmergencyStop )
      Contact( "Axis05_U1_Status".internalEvent )
   END_RUNG wire#w3
   // the same network as SCL:
   #LDrvSafe_SinaTlg903ControlAxis05_U1(STO := true,   // "LDrvSafe_SinaTlg903Control"
                           SS1 := "F-DB_DataFromSafety".EmergencyStop,
                           SS2E := #tEnable_Axis_Move,
                           SLS := NOT (NOT "F-DB_DataFromSafety".DoorsClosed AND "F-DB_DataFromSafety".iKeySettingMode AND "F-DB_DataToSafety".JOG_Mod),
                           SLP := false,
                           SCA := false,
                           ackSafetyFaults := "F-DB_DataToSafety".ResetEmergencyStop AND "Axis05_U1_Status".internalEvent,
                           SinaTlg903Control => "Axis05_U1_Control");
END_REGION

REGION Network 12: Axis06_U2 Status
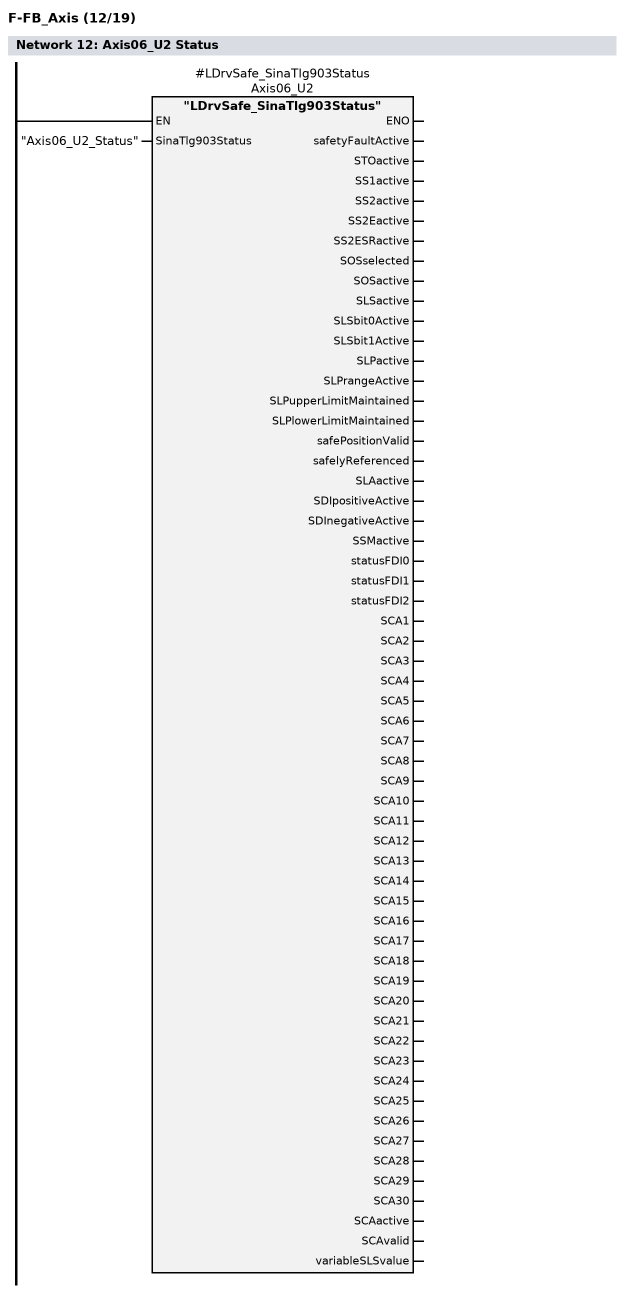
   RUNG wire#powerrail
      #LDrvSafe_SinaTlg903StatusAxis06_U2(SinaTlg903Status := "Axis06_U2_Status", safetyFaultActive =>, STOactive =>, SS1active =>, SS2active =>, SS2Eactive =>, SS2ESRactive =>, SOSselected =>, SOSactive =>, SLSactive =>, SLSbit0Active =>, SLSbit1Active =>, SLPactive =>, SLPrangeActive =>, SLPupperLimitMaintained =>, SLPlowerLimitMaintained =>, safePositionValid =>, safelyReferenced =>, SLAactive =>, SDIpositiveActive =>, SDInegativeActive =>, SSMactive =>, statusFDI0 =>, statusFDI1 =>, statusFDI2 =>, SCA1 =>, SCA2 =>, SCA3 =>, SCA4 =>, SCA5 =>, SCA6 =>, SCA7 =>, SCA8 =>, SCA9 =>, SCA10 =>, SCA11 =>, SCA12 =>, SCA13 =>, SCA14 =>, SCA15 =>, SCA16 =>, SCA17 =>, SCA18 =>, SCA19 =>, SCA20 =>, SCA21 =>, SCA22 =>, SCA23 =>, SCA24 =>, SCA25 =>, SCA26 =>, SCA27 =>, SCA28 =>, SCA29 =>, SCA30 =>, SCAactive =>, SCAvalid =>, variableSLSvalue =>)
   END_RUNG
   // the same network as SCL:
   #LDrvSafe_SinaTlg903StatusAxis06_U2(SinaTlg903Status := "Axis06_U2_Status");   // "LDrvSafe_SinaTlg903Status"
END_REGION

REGION Network 13: Axis06_U2 Control
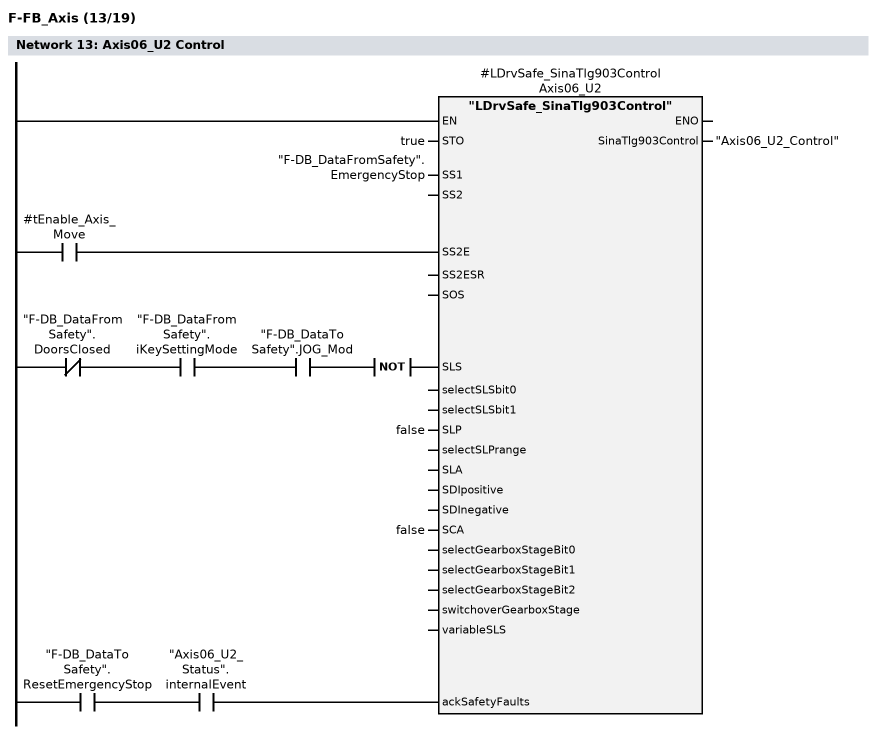
   RUNG wire#powerrail
      #LDrvSafe_SinaTlg903ControlAxis06_U2(SS2E := wire#w1, SLS := wire#w2, ackSafetyFaults := wire#w3, STO := true, SS1 := "F-DB_DataFromSafety".EmergencyStop, SS2 :=, SS2ESR :=, SOS :=, selectSLSbit0 :=, selectSLSbit1 :=, SLP := false, selectSLPrange :=, SLA :=, SDIpositive :=, SDInegative :=, SCA := false, selectGearboxStageBit0 :=, selectGearboxStageBit1 :=, selectGearboxStageBit2 :=, switchoverGearboxStage :=, variableSLS :=, SinaTlg903Control => "Axis06_U2_Control")
   END_RUNG
   RUNG wire#powerrail
      Contact( #tEnable_Axis_Move )
   END_RUNG wire#w1
   RUNG wire#powerrail
      I_Contact( "F-DB_DataFromSafety".DoorsClosed )
      Contact( "F-DB_DataFromSafety".iKeySettingMode )
      Contact( "F-DB_DataToSafety".JOG_Mod )
      Not()
   END_RUNG wire#w2
   RUNG wire#powerrail
      Contact( "F-DB_DataToSafety".ResetEmergencyStop )
      Contact( "Axis06_U2_Status".internalEvent )
   END_RUNG wire#w3
   // the same network as SCL:
   #LDrvSafe_SinaTlg903ControlAxis06_U2(STO := true,   // "LDrvSafe_SinaTlg903Control"
                           SS1 := "F-DB_DataFromSafety".EmergencyStop,
                           SS2E := #tEnable_Axis_Move,
                           SLS := NOT (NOT "F-DB_DataFromSafety".DoorsClosed AND "F-DB_DataFromSafety".iKeySettingMode AND "F-DB_DataToSafety".JOG_Mod),
                           SLP := false,
                           SCA := false,
                           ackSafetyFaults := "F-DB_DataToSafety".ResetEmergencyStop AND "Axis06_U2_Status".internalEvent,
                           SinaTlg903Control => "Axis06_U2_Control");
END_REGION

REGION Network 14: Axis07_V Status
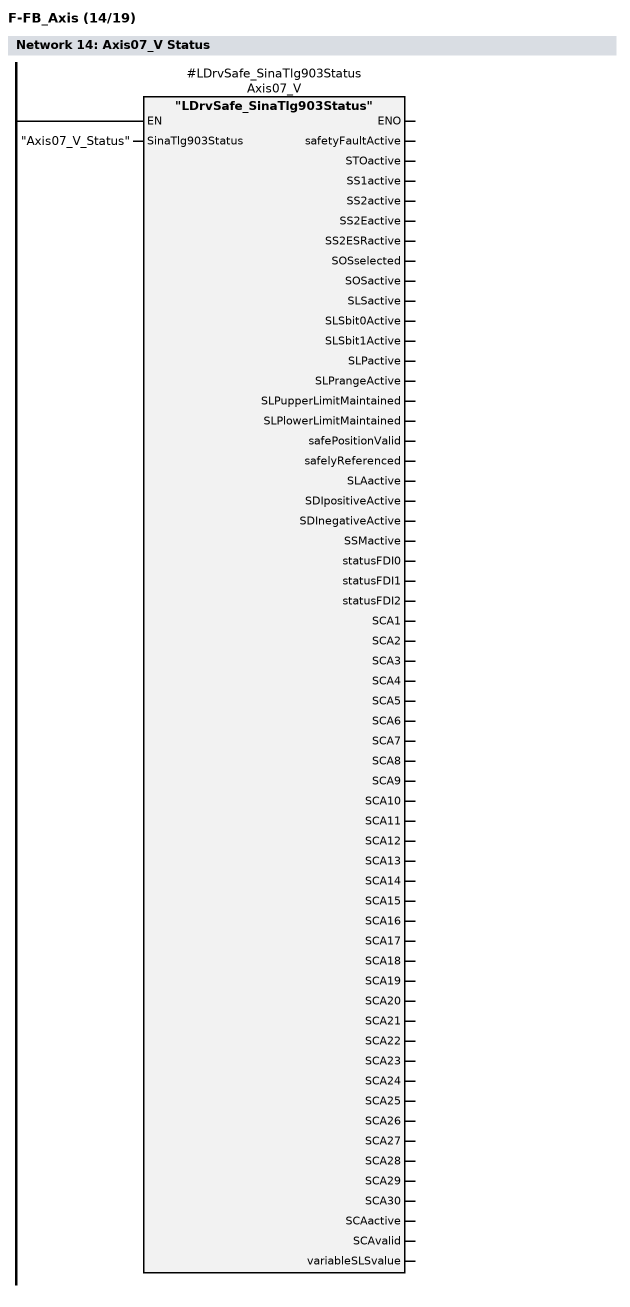
   RUNG wire#powerrail
      #LDrvSafe_SinaTlg903StatusAxis07_V(SinaTlg903Status := "Axis07_V_Status", safetyFaultActive =>, STOactive =>, SS1active =>, SS2active =>, SS2Eactive =>, SS2ESRactive =>, SOSselected =>, SOSactive =>, SLSactive =>, SLSbit0Active =>, SLSbit1Active =>, SLPactive =>, SLPrangeActive =>, SLPupperLimitMaintained =>, SLPlowerLimitMaintained =>, safePositionValid =>, safelyReferenced =>, SLAactive =>, SDIpositiveActive =>, SDInegativeActive =>, SSMactive =>, statusFDI0 =>, statusFDI1 =>, statusFDI2 =>, SCA1 =>, SCA2 =>, SCA3 =>, SCA4 =>, SCA5 =>, SCA6 =>, SCA7 =>, SCA8 =>, SCA9 =>, SCA10 =>, SCA11 =>, SCA12 =>, SCA13 =>, SCA14 =>, SCA15 =>, SCA16 =>, SCA17 =>, SCA18 =>, SCA19 =>, SCA20 =>, SCA21 =>, SCA22 =>, SCA23 =>, SCA24 =>, SCA25 =>, SCA26 =>, SCA27 =>, SCA28 =>, SCA29 =>, SCA30 =>, SCAactive =>, SCAvalid =>, variableSLSvalue =>)
   END_RUNG
   // the same network as SCL:
   #LDrvSafe_SinaTlg903StatusAxis07_V(SinaTlg903Status := "Axis07_V_Status");   // "LDrvSafe_SinaTlg903Status"
END_REGION

REGION Network 15: Axis07_V Control
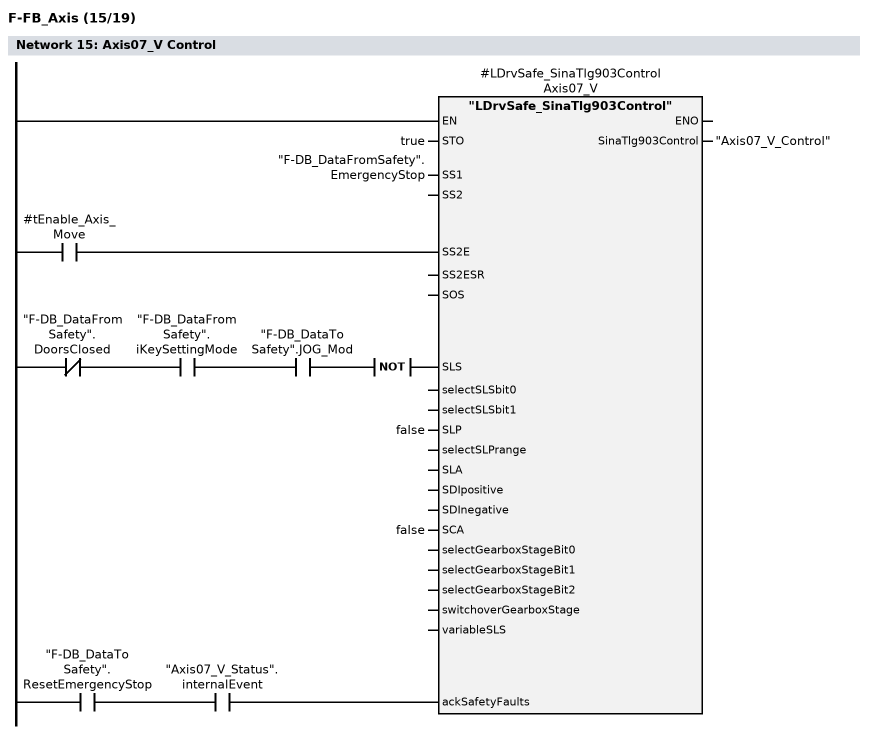
   RUNG wire#powerrail
      #LDrvSafe_SinaTlg903ControlAxis07_V(SS2E := wire#w1, SLS := wire#w2, ackSafetyFaults := wire#w3, STO := true, SS1 := "F-DB_DataFromSafety".EmergencyStop, SS2 :=, SS2ESR :=, SOS :=, selectSLSbit0 :=, selectSLSbit1 :=, SLP := false, selectSLPrange :=, SLA :=, SDIpositive :=, SDInegative :=, SCA := false, selectGearboxStageBit0 :=, selectGearboxStageBit1 :=, selectGearboxStageBit2 :=, switchoverGearboxStage :=, variableSLS :=, SinaTlg903Control => "Axis07_V_Control")
   END_RUNG
   RUNG wire#powerrail
      Contact( #tEnable_Axis_Move )
   END_RUNG wire#w1
   RUNG wire#powerrail
      I_Contact( "F-DB_DataFromSafety".DoorsClosed )
      Contact( "F-DB_DataFromSafety".iKeySettingMode )
      Contact( "F-DB_DataToSafety".JOG_Mod )
      Not()
   END_RUNG wire#w2
   RUNG wire#powerrail
      Contact( "F-DB_DataToSafety".ResetEmergencyStop )
      Contact( "Axis07_V_Status".internalEvent )
   END_RUNG wire#w3
   // the same network as SCL:
   #LDrvSafe_SinaTlg903ControlAxis07_V(STO := true,   // "LDrvSafe_SinaTlg903Control"
                           SS1 := "F-DB_DataFromSafety".EmergencyStop,
                           SS2E := #tEnable_Axis_Move,
                           SLS := NOT (NOT "F-DB_DataFromSafety".DoorsClosed AND "F-DB_DataFromSafety".iKeySettingMode AND "F-DB_DataToSafety".JOG_Mod),
                           SLP := false,
                           SCA := false,
                           ackSafetyFaults := "F-DB_DataToSafety".ResetEmergencyStop AND "Axis07_V_Status".internalEvent,
                           SinaTlg903Control => "Axis07_V_Control");
END_REGION

REGION Network 16: Axis08_W Status
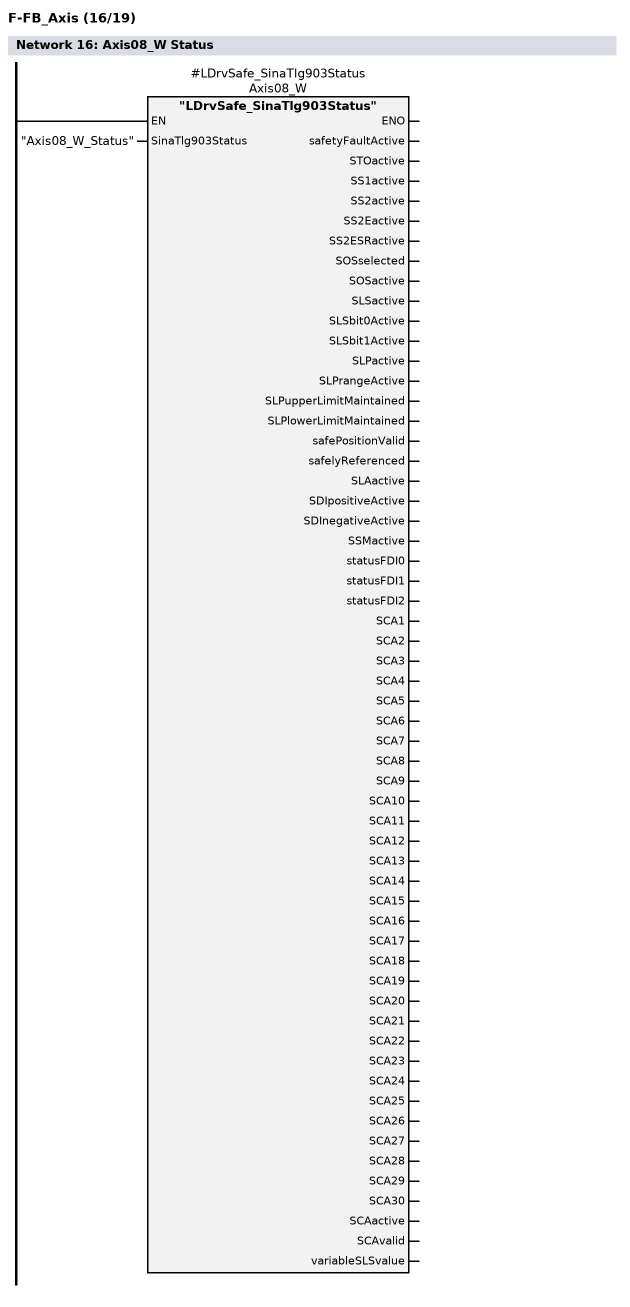
   RUNG wire#powerrail
      #LDrvSafe_SinaTlg903StatusAxis08_W(SinaTlg903Status := "Axis08_W_Status", safetyFaultActive =>, STOactive =>, SS1active =>, SS2active =>, SS2Eactive =>, SS2ESRactive =>, SOSselected =>, SOSactive =>, SLSactive =>, SLSbit0Active =>, SLSbit1Active =>, SLPactive =>, SLPrangeActive =>, SLPupperLimitMaintained =>, SLPlowerLimitMaintained =>, safePositionValid =>, safelyReferenced =>, SLAactive =>, SDIpositiveActive =>, SDInegativeActive =>, SSMactive =>, statusFDI0 =>, statusFDI1 =>, statusFDI2 =>, SCA1 =>, SCA2 =>, SCA3 =>, SCA4 =>, SCA5 =>, SCA6 =>, SCA7 =>, SCA8 =>, SCA9 =>, SCA10 =>, SCA11 =>, SCA12 =>, SCA13 =>, SCA14 =>, SCA15 =>, SCA16 =>, SCA17 =>, SCA18 =>, SCA19 =>, SCA20 =>, SCA21 =>, SCA22 =>, SCA23 =>, SCA24 =>, SCA25 =>, SCA26 =>, SCA27 =>, SCA28 =>, SCA29 =>, SCA30 =>, SCAactive =>, SCAvalid =>, variableSLSvalue =>)
   END_RUNG
   // the same network as SCL:
   #LDrvSafe_SinaTlg903StatusAxis08_W(SinaTlg903Status := "Axis08_W_Status");   // "LDrvSafe_SinaTlg903Status"
END_REGION

REGION Network 17: Axis08_W Control
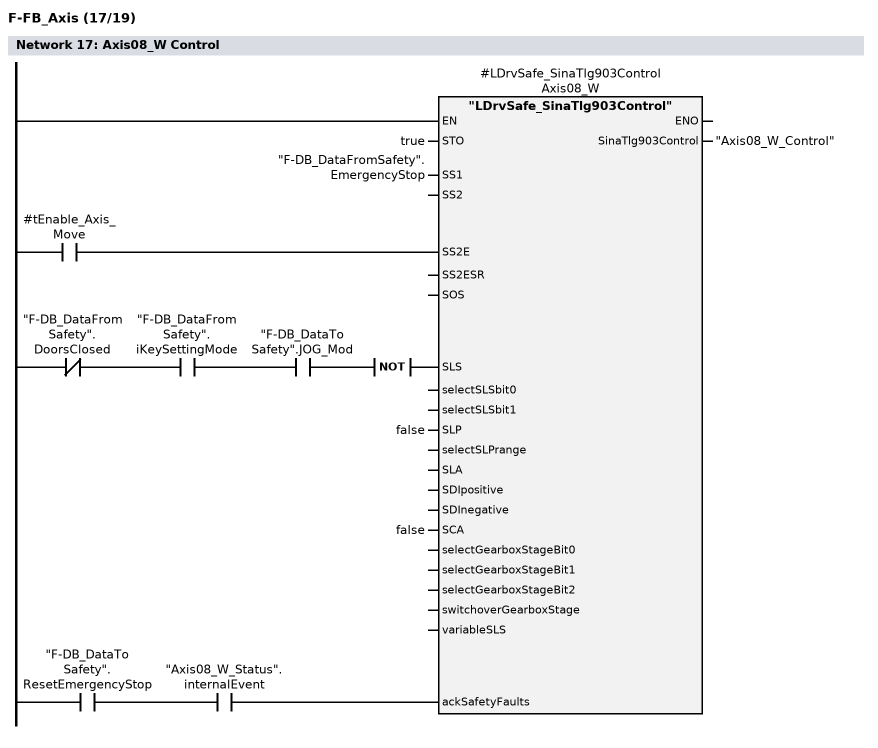
   RUNG wire#powerrail
      #LDrvSafe_SinaTlg903ControlAxis08_W(SS2E := wire#w1, SLS := wire#w2, ackSafetyFaults := wire#w3, STO := true, SS1 := "F-DB_DataFromSafety".EmergencyStop, SS2 :=, SS2ESR :=, SOS :=, selectSLSbit0 :=, selectSLSbit1 :=, SLP := false, selectSLPrange :=, SLA :=, SDIpositive :=, SDInegative :=, SCA := false, selectGearboxStageBit0 :=, selectGearboxStageBit1 :=, selectGearboxStageBit2 :=, switchoverGearboxStage :=, variableSLS :=, SinaTlg903Control => "Axis08_W_Control")
   END_RUNG
   RUNG wire#powerrail
      Contact( #tEnable_Axis_Move )
   END_RUNG wire#w1
   RUNG wire#powerrail
      I_Contact( "F-DB_DataFromSafety".DoorsClosed )
      Contact( "F-DB_DataFromSafety".iKeySettingMode )
      Contact( "F-DB_DataToSafety".JOG_Mod )
      Not()
   END_RUNG wire#w2
   RUNG wire#powerrail
      Contact( "F-DB_DataToSafety".ResetEmergencyStop )
      Contact( "Axis08_W_Status".internalEvent )
   END_RUNG wire#w3
   // the same network as SCL:
   #LDrvSafe_SinaTlg903ControlAxis08_W(STO := true,   // "LDrvSafe_SinaTlg903Control"
                           SS1 := "F-DB_DataFromSafety".EmergencyStop,
                           SS2E := #tEnable_Axis_Move,
                           SLS := NOT (NOT "F-DB_DataFromSafety".DoorsClosed AND "F-DB_DataFromSafety".iKeySettingMode AND "F-DB_DataToSafety".JOG_Mod),
                           SLP := false,
                           SCA := false,
                           ackSafetyFaults := "F-DB_DataToSafety".ResetEmergencyStop AND "Axis08_W_Status".internalEvent,
                           SinaTlg903Control => "Axis08_W_Control");
END_REGION

REGION Network 18: Axis09_ZL Status
